fb_stat(xIN_Enable  := enIN_State = enState.StateAUTO,
        xIN_Waiting := fb_Pnp.xOUT_Wait,
        xIN_Running := (fb_Pnp.iOUT_Step >= ST180_Pnp_e.START) AND
                       (fb_Pnp.iOUT_Step <= ST180_Pnp_e.DONE),
        // Since we use a mover system, a cycle is done when we are waiting on a mover
        xIN_Done := fb_Pnp.iOUT_Step = ST180_Pnp_e.waitOnMover);

(*******************************************************************)
(* Mover reset flags *)
(*******************************************************************)

(*******************************************************************)
(* OUTPUT *)
(*******************************************************************)
xOUT_InitDone := fb_Pnp.xOUT_InitDone;
xOUT_Ready    := fb_Pnp.xOUT_Ready;
xOUT_Done     := fb_Pnp.xOUT_Done;
xOUT_ErrFlag  := fb_Pnp.xOUT_ErrFlag;
xOUT_Wait     := fb_Pnp.xOUT_Wait;
xOUT_AlarmST  := xOUT_ErrFlag;

(*******************************************************************)
(* Bausteinaufruf Error Station *)
(*******************************************************************)
// POU_ERR_VORLAGE(xIN_QUIT:=xIN_Quit , pstrArIN_ALARM:=ADR(HMI.strArALARM[1]));

(* % of completion of the process *)
PROPERTY iCompletionPC : INT
GET
iCompletionPC := THIS^.fb_Pnp.iOUT_ProcessCompletion;
END_GET
END_PROPERTY

PROPERTY ProcessExecution : ProcessExecution_e
GET
ProcessExecution := THIS^._ProcessExecution;
END_GET
SET
THIS^._ProcessExecution := ProcessExecution;
END_SET
END_PROPERTY

PROPERTY xBusy : BOOL
GET
xBusy := THIS^.fb_Pnp.xOUT_Busy;
END_GET
SET
END_SET
END_PROPERTY

PROPERTY xDone : BOOL
GET
xDone := THIS^.fb_Pnp.xOUT_Ready OR THIS^.fb_Pnp.xOUT_Done;
END_GET
END_PROPERTY

PROPERTY xMoverPathFree : BOOL
GET
xMoverPathFree := THIS^.fb_Pnp.xOUT_MoverFree OR THIS^.fb_Pnp.xOUT_Ready OR THIS^.fb_Pnp.xOUT_Done;
END_GET
END_PROPERTY

PROPERTY xMoverShouldLeave : BOOL
GET
xMoverShouldLeave := THIS^.fb_Pnp.iOUT_Step = ST180_Pnp_e.SYNC_MOVER_LEAVE;
END_GET
END_PROPERTY

END_FUNCTION_BLOCK

// ---- POUs/20_AUTO/ST180/FB_ABL_180_Pnp.TcPOU
FUNCTION_BLOCK FB_ABL_180_Pnp
(****************************************************************************************)
(*	TITEL				laden kristall- Modul	    										*)
(*	Status				ungetestet                         								*)
(*	Beschrieb:			Ablaufbeschreibung												*)
(*																						*)
(*	Steps:	self-explained using enum													*)
(***********************************Revisionen*******************************************)
(*	see github blames																	*)
(****************************************************************************************)

VAR_INPUT
    xIN_Reset       : BOOL;          // Schrittkette zurücksetzen 
    xIN_Init        : BOOL;          // Initialisieren
    xIN_Quit        : BOOL;          // Fehler quittieren 
    xIN_Start       : BOOL;          // Startbefehl
    xIN_Sperre      : BOOL;          // FB Sperren 
    xIN_NextStep    : BOOL;          // Nächsten Schritt ausführen 
    xIN_AlarmAktiv  : BOOL;          // Anlage hat Alarm
    xIN_DryCycle    : BOOL;          // Fahren ohne Teile
    xIN_RestartCYCL : BOOL;          // Zyklus erneut starten im STEP: END: LEERFAHREN
    enIN_State      : enState;       // Status Anlage
    tIN_Timeout     : TIME := T#10s; // Timout

    pxFG_Freigabe : POINTER TO BOOL; //Freigabe von Station

    // Application specific
    Mover              : REFERENCE TO FB_Mover;
    xIN_PceReadyToPick : BOOL; // the piece(s) is/are ready to picked
END_VAR
VAR_OUTPUT
    (* standart Ausgänge *)
    xOUT_ErrFlag  : BOOL;        // Error Flag 
    xOUT_Busy     : BOOL;        // Baustein befindet sich im Ablauf 
    xOUT_Done     : BOOL;        // Baustein hat den Ablauf beendet 		
    xOUT_Ready    : BOOL;        // Ready to begin: should be the same state as done	
    xOUT_Timeout  : BOOL;        // Timeout FB 
    xOUT_InitDone : BOOL;        // initialisierung fertig
    xOUT_Wait     : BOOL;        // Wartet auf Bedingung
    iOUT_Step     : ST180_Pnp_e; // Aktueller Schritt 
    sOUT_Step     : STRING;      // Aktueller Schritt but in string format
    bOUT_Error    : BYTE;        // Fehlernummer

    iOUT_ProcessCompletion : INT;  //process completion: express in % (0-100)
    xOUT_MoverFree         : BOOL; // The mover is free to move

END_VAR
VAR
    (* Standard *)
    (* Schritt *)
    iLastStep : ST180_Pnp_e; // Merker letzter Schritt 
    iPreStep  : ST180_Pnp_e; // Schritt zurück nach Alarm 
    iAktStep  : ST180_Pnp_e; // aktueller Schritt

    // Trigger Starten 
    rtSTART : R_TRIG;
    // Timer TimeOut 
    TON_Timeout : TON;

    (* Bausteine *)

    (* Spezial *)
    fb_axis180_01Y : FB_AxisLM_V1_1;
    fb_axis180_02Z : FB_AxisLM_V1_1;
    fb_axis180_10Z : FB_AxisLM_V1_1;

    fb_PnpHorAxis    : FB_LinearMotionMan;
    fb_PnpVerAxis_02 : FB_LinearMotionMan;
    fb_PnpVerAxis_10 : FB_LinearMotionMan;

    fb_simu_axis180_01Y : FB_Simu_AxisLM_V1_1;
    fb_simu_axis180_02Z : FB_Simu_AxisLM_V1_1;
    fb_simu_axis180_10Z : FB_Simu_AxisLM_V1_1;

    fb_griperLeft    : FB_ZylMo2El_V2_1;
    fb_griperRight   : FB_ZylMo2El_V2_1;
    simu_griperLeft  : FB_Simu_Zyl2Pos;
    simu_griperRight : FB_Simu_Zyl2Pos;
    fb_clampLeft     : FB_ZylMo2El_V2_1;
    fb_clampRight    : FB_ZylMo2El_V2_1;
    simu_clampLeft   : FB_Simu_Zyl2Pos;
    simu_clampRight  : FB_Simu_Zyl2Pos;

END_VAR
VAR CONSTANT
    PNP_SIMULATION : BOOL := FALSE; // Set to TRUE to simulate this part of the program
END_VAR

(*******************************************************************)
(* Trigger  *)
(*******************************************************************)
(* Zurücksetzen *)
IF xIN_RESET THEN
    iPreStep  := ST180_Pnp_e.RESET;
    iOUT_Step := ST180_Pnp_e.RESET;
END_IF;

(* Error Quittieren *)
IF (bOUT_Error <> 0) AND xIN_Quit THEN
    xOUT_ErrFlag := FALSE;
    bOUT_Error   := 0;
    iOUT_Step    := iPreStep;
END_IF;

(*******************************************************************)
(* Timer *)
(*******************************************************************)
TON_Timeout(IN := xIN_NextStep AND (iLastStep = iOUT_Step) (*todo FG *) ,
            PT := tIN_Timeout);

(*******************************************************************)
(* Bausteine *)
(*******************************************************************)
fb_PnpHorAxis(config          := _20_AUTO.recipe.linearAxis[LinearAxis_e.ST180_01Y],
              xIN_Init        := enIN_State = enState.StateINIT,
              xIN_Reset       := xIN_Reset,
              lrIN_CurrPos    := fb_axis180_01Y.rOUT_ActPos,
              lrIN_Delta_mm   := 1.0,
              iIN_CurrentStep := iOUT_Step,
              iIN_moveNumber  := ST180_PnpHorPos_e._max);

fb_simu_axis180_01Y(xIN_Enable          := PNP_SIMULATION AND CONST.USE_SIMULATION,
                    bIN_AxisCntr        := fb_axis180_01Y.bOUT_AxisCntr,
                    wIN_AxisState       := ST180_Axis.axis180_01Y.wState,
                    udiIN_HomingTime_ms := 2000,
                    pIN_axisSimu        := ADR(SIMU.axis_ref[Axis_e.ST180_01Y]),
                    pIN_axisHW          := ADR(ST180_Axis.axis180_01Y.axis),
                    rIN_PosActual       := ST180_Axis.axis180_01Y.rActPos,
                    rIN_PosMax          := ST180_Axis.const180_01Y.POS_MAX,
                    rIN_PosMin          := ST180_Axis.const180_01Y.POS_MIN,
                    rIN_PixMax          := 100,
                    rIN_PixMin          := 0);

fb_axis180_01Y(enIN_State       := enIN_State,
               parIN_Buttons    := ADR(AXIS.btTeachArAxis[Axis_e.ST180_01Y]),
               xIN_DisButtons   := FALSE,
               xIN_Quit         := xIN_Quit,
               xIN_PARAMok      := TRUE, (*TODO*)
               xIN_FREE         := TRUE,
               xIN_FREE_HOME    := TRUE,
               rIN_POSMIN       := ST180_Axis.const180_01Y.POS_MIN,
               rIN_POSMAX       := ST180_Axis.const180_01Y.POS_MAX,
               rIN_VELOMAX      := ST180_Axis.const180_01Y.VELO_MAX,
               rIN_VELOMANU     := ST180_Axis.const180_01Y.VELO_MANU,
               rIN_VELOOPEN     := ST180_Axis.const180_01Y.VELO_MANU / 4,
               rIN_JogInc       := AXIS.rTeachIncAxis,
               xIN_Execute      := fb_PnpHorAxis.xOUT_Execute,
               xIN_Relative     := FALSE,
               xIN_STOP         := FALSE,
               xIN_OFF          := FALSE,
               rIN_Position     := TO_REAL(fb_PnpHorAxis.OUT_MoveProfile.lrPosition),
               rIN_Velocity     := TO_REAL(fb_PnpHorAxis.OUT_MoveProfile.lrVelocity),
               rIN_Acceleration := TO_REAL(fb_PnpHorAxis.OUT_MoveProfile.lrAccel),
               rIN_Deceleration := TO_REAL(fb_PnpHorAxis.OUT_MoveProfile.lrDecel),
               rIN_Jerk         := TO_REAL(fb_PnpHorAxis.OUT_MoveProfile.lrJerk),
               rIN_PosManu      := TO_REAL(_20_AUTO.recipe.linearAxis[LinearAxis_e.ST180_01Y]
                                               .movesList[AXIS.bTeachPos[Axis_e.ST180_01Y]].lrPosition),
               rIN_VeloJogManu := TO_REAL(Axis.rJogVelo_pc),
               xIN_Home        := ST180_Pnp_e.Init_HomeHorizontal = iOUT_Step,
               xIN_Reset       := (ST180_Pnp_e.RESET = iOUT_Step) OR xIN_Reset,
               // The simu fb gives the hardware state when we are not in simu
               wAxisState    := fb_simu_axis180_01Y.wOUT_AxisState,
               bOUT_AxisCntr => st180_axis.axis180_01Y.bCtrlHi,
               rOUT_ActPos   => st180_axis.axis180_01Y.rActPos,
               axisIN_REF    := fb_simu_axis180_01Y.pOUT_axisRef^);

fb_PnpVerAxis_02(config          := _20_AUTO.recipe.linearAxis[LinearAxis_e.ST180_02Z],
                 xIN_Init        := enIN_State = enState.StateINIT,
                 xIN_Reset       := xIN_Reset,
                 lrIN_CurrPos    := fb_axis180_02Z.rOUT_ActPos,
                 lrIN_Delta_mm   := 2.50,
                 iIN_CurrentStep := iOUT_Step,
                 iIN_moveNumber  := ST180_PnpVerPos_e._max);

fb_simu_axis180_02Z(xIN_Enable          := PNP_SIMULATION AND CONST.USE_SIMULATION,
                    bIN_AxisCntr        := fb_axis180_02Z.bOUT_AxisCntr,
                    wIN_AxisState       := ST180_Axis.axis180_02Z.wState,
                    udiIN_HomingTime_ms := 2000,
                    pIN_axisSimu        := ADR(SIMU.axis_ref[Axis_e.ST180_02Z]),
                    pIN_axisHW          := ADR(ST180_Axis.axis180_02Z.axis),
                    rIN_PosActual       := ST180_Axis.axis180_02Z.rActPos,
                    rIN_PosMax          := ST180_Axis.const180_02Z.POS_MAX,
                    rIN_PosMin          := ST180_Axis.const180_02Z.POS_MIN,
                    rIN_PixMax          := 100,
                    rIN_PixMin          := 0);

fb_axis180_02Z(enIN_State       := enIN_State,
               parIN_Buttons    := ADR(AXIS.btTeachArAxis[Axis_e.ST180_02Z]),
               xIN_DisButtons   := FALSE,
               xIN_Quit         := xIN_Quit,
               xIN_PARAMok      := TRUE,
               xIN_FREE         := TRUE,
               xIN_FREE_HOME    := TRUE,
               rIN_POSMIN       := ST180_Axis.const180_02Z.POS_MIN,
               rIN_POSMAX       := ST180_Axis.const180_02Z.POS_MAX,
               rIN_VELOMAX      := ST180_Axis.const180_02Z.VELO_MAX,
               rIN_VELOMANU     := ST180_Axis.const180_02Z.VELO_MANU,
               rIN_VELOOPEN     := ST180_Axis.const180_02Z.POS_MAX / 4,
               rIN_JogInc       := AXIS.rTeachIncAxis,
               xIN_Execute      := fb_PnpVerAxis_02.xOUT_Execute,
               xIN_Relative     := FALSE,
               xIN_STOP         := FALSE,
               xIN_OFF          := FALSE,
               rIN_Position     := TO_REAL(fb_PnpVerAxis_02.OUT_MoveProfile.lrPosition),
               rIN_Velocity     := TO_REAL(fb_PnpVerAxis_02.OUT_MoveProfile.lrVelocity),
               rIN_Acceleration := TO_REAL(fb_PnpVerAxis_02.OUT_MoveProfile.lrAccel),
               rIN_Deceleration := TO_REAL(fb_PnpVerAxis_02.OUT_MoveProfile.lrDecel),
               rIN_Jerk         := TO_REAL(fb_PnpVerAxis_02.OUT_MoveProfile.lrJerk),
               rIN_PosManu      := TO_REAL(_20_AUTO.recipe.linearAxis[LinearAxis_e.ST180_02Z]
                                               .movesList[AXIS.bTeachPos[Axis_e.ST180_02Z]].lrPosition),
               rIN_VeloJogManu := TO_REAL(Axis.rJogVelo_pc),
               xIN_Home        := ST180_Pnp_e.Init_HomeVertical_02 = iOUT_Step,
               xIN_Reset       := (ST180_Pnp_e.RESET = iOUT_Step) OR xIN_Reset,
               wAxisState      := fb_simu_axis180_02Z.wOUT_AxisState,
               bOUT_AxisCntr   => ST180_Axis.axis180_02Z.bCtrlHi,
               rOUT_ActPos     => ST180_Axis.axis180_02Z.rActPos,
               axisIN_REF      := fb_simu_axis180_02Z.pOUT_axisRef^);

fb_PnpVerAxis_10(config          := _20_AUTO.recipe.linearAxis[LinearAxis_e.ST180_10Z],
                 xIN_Init        := enIN_State = enState.StateINIT,
                 xIN_Reset       := xIN_Reset,
                 lrIN_CurrPos    := fb_axis180_10Z.rOUT_ActPos,
                 lrIN_Delta_mm   := 1.0,
                 iIN_CurrentStep := iOUT_Step,
                 iIN_moveNumber  := ST180_PnpVerPos_e._max);

fb_simu_axis180_10Z(xIN_Enable          := PNP_SIMULATION AND CONST.USE_SIMULATION,
                    bIN_AxisCntr        := fb_axis180_10Z.bOUT_AxisCntr,
                    wIN_AxisState       := ST180_Axis.axis180_10Z.wState,
                    udiIN_HomingTime_ms := 2000,
                    pIN_axisSimu        := ADR(SIMU.axis_ref[Axis_e.ST180_10Z]),
                    pIN_axisHW          := ADR(ST180_Axis.axis180_10Z.axis),
                    rIN_PosActual       := ST180_Axis.axis180_10Z.rActPos,
                    rIN_PosMax          := ST180_Axis.const180_10Z.POS_MAX,
                    rIN_PosMin          := ST180_Axis.const180_10Z.POS_MIN,
                    rIN_PixMax          := 100,
                    rIN_PixMin          := 0);

fb_axis180_10Z(enIN_State       := enIN_State,
               parIN_Buttons    := ADR(AXIS.btTeachArAxis[Axis_e.ST180_10Z]),
               xIN_DisButtons   := FALSE,
               xIN_Quit         := xIN_Quit,
               xIN_PARAMok      := TRUE,
               xIN_FREE         := TRUE,
               xIN_FREE_HOME    := TRUE,
               rIN_POSMIN       := ST180_Axis.const180_10Z.POS_MIN,
               rIN_POSMAX       := ST180_Axis.const180_10Z.POS_MAX,
               rIN_VELOMAX      := ST180_Axis.const180_10Z.VELO_MAX,
               rIN_VELOMANU     := ST180_Axis.const180_10Z.VELO_MANU,
               rIN_VELOOPEN     := ST180_Axis.const180_10Z.POS_MAX / 4,
               rIN_JogInc       := AXIS.rTeachIncAxis,
               xIN_Execute      := fb_PnpVerAxis_10.xOUT_Execute,
               xIN_Relative     :=,
               xIN_STOP         :=,
               xIN_OFF          :=,
               rIN_Position     := TO_REAL(fb_PnpVerAxis_10.OUT_MoveProfile.lrPosition),
               rIN_Velocity     := TO_REAL(fb_PnpVerAxis_10.OUT_MoveProfile.lrVelocity),
               rIN_Acceleration := TO_REAL(fb_PnpVerAxis_10.OUT_MoveProfile.lrAccel),
               rIN_Deceleration := TO_REAL(fb_PnpVerAxis_10.OUT_MoveProfile.lrDecel),
               rIN_Jerk         := TO_REAL(fb_PnpVerAxis_10.OUT_MoveProfile.lrJerk),
               rIN_PosManu      := TO_REAL(_20_AUTO.recipe.linearAxis[LinearAxis_e.ST180_10Z]
                                               .movesList[AXIS.bTeachPos[Axis_e.ST180_10Z]].lrPosition),
               rIN_VeloJogManu := TO_REAL(Axis.rJogVelo_pc),
               xIN_Home        := ST180_Pnp_e.Init_HomeVertical_10 = iOUT_Step,
               xIN_Reset       := (ST180_Pnp_e.RESET = iOUT_Step) OR xIN_Reset,
               wAxisState      := fb_simu_axis180_10Z.wOUT_AxisState,
               bOUT_AxisCntr   => ST180_Axis.axis180_10Z.bCtrlHi,
               rOUT_ActPos     => ST180_Axis.axis180_10Z.rActPos,
               axisIN_REF      := fb_simu_axis180_10Z.pOUT_axisRef^);

//////////////////////////////////
fb_griperLeft(xIN_Reset    := xIN_Reset OR (ST180_Pnp_e.RESET = iOUT_Step),
              xIN_Quit     := xIN_Quit,
              xIN_Manu     := enState.StateMANU = enIN_State,
              pbtIN_Button := ADR(HMI.btManuCylinders[StationList_e.ST180][1]),
              xIN_GS       := simu_griperLeft.xOUT_inGS,
              xIN_AS       := simu_griperLeft.xOUT_inAS,
              xIN_FREE     := TRUE,
              xINtoGS      := _20_AUTO.recipe.st180.xUseVerLeft AND ST180_Pnp_e.close_griper_pick_piece = iOUT_Step,
              xINtoAS      := ST180_Pnp_e.open_griper_put_piece = iOUT_Step,
              tIN_ErrAS    := DINT_TO_TIME(_20_AUTO.recipe.cylinder2Pos[StationList_e.ST180]
                                               [ST180_Cylinders_e.Greifer_Patrone_Links].toAS_alarm_time),
              tIN_ErrGS := DINT_TO_TIME(_20_AUTO.recipe.cylinder2Pos[StationList_e.ST180]
                                            [ST180_Cylinders_e.Greifer_Patrone_Links].toGS_alarm_time),
              tIN_WaitAS := DINT_TO_TIME(_20_AUTO.recipe.cylinder2Pos[StationList_e.ST180]
                                             [ST180_Cylinders_e.Greifer_Patrone_Links].toAS_wait_time),
              tIN_WaitGS := DINT_TO_TIME(_20_AUTO.recipe.cylinder2Pos[StationList_e.ST180]
                                             [ST180_Cylinders_e.Greifer_Patrone_Links].toGS_wait_time));

simu_griperLeft(xIN_Enable := PNP_SIMULATION AND CONST.USE_SIMULATION,
                xIN_inGS   := IO_BOX.I9100_ST180_greifer_patrone_links_zu,
                xIN_inAS   := IO_BOX.I9101_ST180_greifer_patrone_links_offen,
                xIN_valve  := fb_griperLeft.xOUT_VALVE,
                tIN_GS_ms  := 200,  //ms
                tIN_AS_ms  := 200); //ms

fb_griperRight(xIN_Reset    := xIN_Reset OR (ST180_Pnp_e.RESET = iOUT_Step),
               xIN_Quit     := xIN_Quit,
               xIN_Manu     := enState.StateMANU = enIN_State,
               pbtIN_Button := ADR(HMI.btManuCylinders[StationList_e.ST180][2]),
               xIN_GS       := simu_griperRight.xOUT_inGS,
               xIN_AS       := simu_griperRight.xOUT_inAS,
               xIN_FREE     := TRUE,
               xINtoGS      := _20_AUTO.recipe.st180.xUseVerRight AND ST180_Pnp_e.close_griper_pick_piece = iOUT_Step,
               xINtoAS      := ST180_Pnp_e.open_griper_put_piece = iOUT_Step,
               tIN_ErrAS    := DINT_TO_TIME(_20_AUTO.recipe.cylinder2Pos[StationList_e.ST180]
                                                [ST180_Cylinders_e.Greifer_Patrone_Rechts].toAS_alarm_time),
               tIN_ErrGS := DINT_TO_TIME(_20_AUTO.recipe.cylinder2Pos[StationList_e.ST180]
                                             [ST180_Cylinders_e.Greifer_Patrone_Rechts].toGS_alarm_time),
               tIN_WaitAS := DINT_TO_TIME(_20_AUTO.recipe.cylinder2Pos[StationList_e.ST180]
                                              [ST180_Cylinders_e.Greifer_Patrone_Rechts].toAS_wait_time),
               tIN_WaitGS := DINT_TO_TIME(_20_AUTO.recipe.cylinder2Pos[StationList_e.ST180]
                                              [ST180_Cylinders_e.Greifer_Patrone_Rechts].toGS_wait_time));

simu_griperRight(xIN_Enable := PNP_SIMULATION AND CONST.USE_SIMULATION,
                 xIN_inGS   := IO_BOX.I9102_ST180_greifer_patrone_rechts_zu,
                 xIN_inAS   := IO_BOX.I9103_ST180_greifer_patrone_rechts_offen,
                 xIN_valve  := fb_griperRight.xOUT_VALVE,
                 tIN_GS_ms  := 200,  //ms
                 tIN_AS_ms  := 200); //ms

fb_clampLeft(xIN_Reset    := xIN_Reset OR (ST180_Pnp_e.RESET = iOUT_Step),
             xIN_Quit     := xIN_Quit,
             xIN_Manu     := enState.StateMANU = enIN_State,
             pbtIN_Button := ADR(HMI.btManuCylinders[StationList_e.ST180][3]),
             xIN_GS       := simu_clampLeft.xOUT_inGS,
             xIN_AS       := simu_clampLeft.xOUT_inAS,
             xIN_FREE     := TRUE,
             xINtoGS      := ST180_Pnp_e.clamp_up_to_rest_position = iOUT_Step,
             xINtoAS      := _20_AUTO.recipe.st180.xUseVerLeft AND
                             (ST180_Pnp_e.clamp_down_maintain_piece = iOUT_Step),
             tIN_ErrAS := DINT_TO_TIME(_20_AUTO.recipe.cylinder2Pos[StationList_e.ST180]
                                           [ST180_Cylinders_e.Niederhalter_Deckel_Links].toAS_alarm_time),
             tIN_ErrGS := DINT_TO_TIME(_20_AUTO.recipe.cylinder2Pos[StationList_e.ST180]
                                           [ST180_Cylinders_e.Niederhalter_Deckel_Links].toGS_alarm_time),
             tIN_WaitAS := DINT_TO_TIME(_20_AUTO.recipe.cylinder2Pos[StationList_e.ST180]
                                            [ST180_Cylinders_e.Niederhalter_Deckel_Links].toAS_wait_time),
             tIN_WaitGS := DINT_TO_TIME(_20_AUTO.recipe.cylinder2Pos[StationList_e.ST180]
                                            [ST180_Cylinders_e.Niederhalter_Deckel_Links].toGS_wait_time));

simu_clampLeft(xIN_Enable := PNP_SIMULATION AND CONST.USE_SIMULATION,
               xIN_inGS   := IO_BOX.I9104_ST180_niederhalter_deckel_links_oben,
               xIN_inAS   := NOT IO_BOX.I9104_ST180_niederhalter_deckel_links_oben,
               xIN_valve  := fb_clampLeft.xOUT_VALVE,
               tIN_GS_ms  := 200,  //ms
               tIN_AS_ms  := 200); //ms

fb_clampRight(xIN_Reset    := xIN_Reset OR (ST180_Pnp_e.RESET = iOUT_Step),
              xIN_Quit     := xIN_Quit,
              xIN_Manu     := enState.StateMANU = enIN_State,
              pbtIN_Button := ADR(HMI.btManuCylinders[StationList_e.ST180][4]),
              xIN_GS       := simu_clampRight.xOUT_inGS,
              xIN_AS       := simu_clampRight.xOUT_inAS,
              xIN_FREE     := TRUE,
              xINtoGS      := ST180_Pnp_e.clamp_up_to_rest_position = iOUT_Step,
              xINtoAS      := _20_AUTO.recipe.st180.xUseVerRight AND
                              (ST180_Pnp_e.clamp_down_maintain_piece = iOUT_Step),
              tIN_ErrAS := DINT_TO_TIME(_20_AUTO.recipe.cylinder2Pos[StationList_e.ST180]
                                            [ST180_Cylinders_e.Niederhalter_Deckel_Rechts].toAS_alarm_time),
              tIN_ErrGS := DINT_TO_TIME(_20_AUTO.recipe.cylinder2Pos[StationList_e.ST180]
                                            [ST180_Cylinders_e.Niederhalter_Deckel_Rechts].toGS_alarm_time),
              tIN_WaitAS := DINT_TO_TIME(_20_AUTO.recipe.cylinder2Pos[StationList_e.ST180]
                                             [ST180_Cylinders_e.Niederhalter_Deckel_Rechts].toAS_wait_time),
              tIN_WaitGS := DINT_TO_TIME(_20_AUTO.recipe.cylinder2Pos[StationList_e.ST180]
                                             [ST180_Cylinders_e.Niederhalter_Deckel_Rechts].toGS_wait_time));

simu_clampRight(xIN_Enable := PNP_SIMULATION AND CONST.USE_SIMULATION,
                xIN_inGS   := IO_BOX.I9106_ST180_niederhalter_deckel_rechts_oben,
                xIN_inAS   := NOT IO_BOX.I9106_ST180_niederhalter_deckel_rechts_oben,
                xIN_valve  := fb_clampRight.xOUT_VALVE,
                tIN_GS_ms  := 200,  // ms
                tIN_AS_ms  := 200); // ms

(*******************************************************************)
(* OUTPUTS *)
(*******************************************************************)
// Error Flag 
xOUT_ErrFlag := (bOUT_Error <> 0) OR (ST180_Pnp_e.ERROR = iOUT_Step);
// Baustein befindet sich im Ablauf 
xOUT_Busy := (iOUT_Step > ST180_Pnp_e.READY) AND (iOUT_Step < ST180_Pnp_e.DONE);
// Baustein hat den Ablauf beendet
xOUT_Done := (iOUT_Step = ST180_Pnp_e.DONE);
// Process ready
xOUT_Ready := (iOUT_Step = ST180_Pnp_e.READY) OR (iOUT_Step = ST180_Pnp_e.hor_move_to_extraction_pipe);
// Timeout FB 				 		
xOUT_Timeout := TON_Timeout.Q;
// Itialisierung fertig			
xOUT_InitDone := (iOUT_Step = ST180_Pnp_e.READY) OR
                 (iOUT_Step = ST180_Pnp_e.hor_move_to_extraction_pipe) OR
                 (iOUT_Step = ST180_Pnp_e.DONE);

// Aktueller Schritt			
iOUT_Step := iOUT_Step; //Im Ablauf gesetzt		
sOUT_Step := TO_STRING(iOUT_Step);
//Fehlernummer	 
bOUT_Error := bOUT_Error; //Im Ablauf/FB gesetzt	
(* Warte (alle Schritte wo auf FG oder Teile gewartet wird) *)
xOUT_Wait := (iOUT_Step = ST180_Pnp_e.DONE) OR
             (iOUT_Step = ST180_Pnp_e.READY) OR
             (iOUT_Step = ST180_Pnp_e.START) OR
             (iOUT_Step = ST180_Pnp_e.waitOnMover) OR
             (iOUT_Step = ST180_Pnp_e.SYNC_MOVER_LEAVE);

xOUT_MoverFree := NOT (iOUT_Step >= ST180_Pnp_e.MOVER_NEEDED_OP AND iOUT_Step < ST180_Pnp_e.MOVER_FREE_OP) AND
                  (iOUT_Step >= ST180_Pnp_e.READY) AND
                  (iOUT_Step < ST180_Pnp_e.ERROR);

iOUT_ProcessCompletion := F_GetPercent_2(iOUT_Step,
                                         ST180_Pnp_e.lift_piece_and_down_to_pick,
                                         ST180_Pnp_e.take_out_piece_and_put_down_lifter,
                                         ST180_Pnp_e.hor_move_to_extraction_pipe,
                                         ST180_Pnp_e.hor_to_track_pos);

// TODO Valve should not be set when we are in simulation !
IO_BOX.Q5400_14_ST180_greifer_patrone_links :=
    fb_griperLeft.xOUT_VALVE AND NOT (PNP_SIMULATION AND CONST.USE_SIMULATION);

IO_BOX.Q5401_14_ST180_greifer_patrone_rechts :=
    fb_griperRight.xOUT_VALVE AND NOT (PNP_SIMULATION AND CONST.USE_SIMULATION);

IO_BOX.Q5402_14_ST180_niederhalter_deckel_links :=
    fb_clampLeft.xOUT_VALVE AND NOT (PNP_SIMULATION AND CONST.USE_SIMULATION);

IO_BOX.Q5403_14_ST180_Niederhalter_deckel_rechts :=
    fb_clampRight.xOUT_VALVE AND NOT (PNP_SIMULATION AND CONST.USE_SIMULATION);

// safety pneumatics
IO_BOX.Q5408_14_ST180_Break_axis_02Z := NOT fb_simu_axis180_02Z.pIN_axisHW^.Status.Error AND
                                        _02_SAFETY.xOUT_ESout AND
                                        _02_SAFETY.xOUT_MonOut AND
                                        NOT (PNP_SIMULATION AND CONST.USE_SIMULATION);

(*******************************************************************)
(* Ablauf *)
(*******************************************************************)

(* Sperren *)
IF xIN_Sperre THEN
    iPreStep  := ST180_Pnp_e.RESET;
    iOUT_Step := ST180_Pnp_e.RESET;
    RETURN;
END_IF;

(* Schritt Merker *)
IF iAktStep <> iOUT_Step THEN
    iLastStep := iAktStep;
    iAktStep  := iOUT_Step;
END_IF

(* START *)
rtSTART(CLK := xIN_Start);

IF 0 = bOUT_Error THEN
    IF fb_axis180_01Y.xOUT_ErrFlag THEN
        bOUT_Error := 11;
    ELSIF fb_axis180_02Z.xOUT_ErrFlag THEN
        bOUT_Error := 12;
    ELSIF fb_axis180_10Z.xOUT_ErrFlag THEN
        bOUT_Error := 13;
    ELSIF fb_griperLeft.xOUT_ErrFlag THEN
        bOUT_Error := 14;
    ELSIF fb_griperRight.xOUT_ErrFlag THEN
        bOUT_Error := 15;
    ELSIF fb_clampLeft.xOUT_ErrFlag THEN
        bOUT_Error := 16;
    ELSIF fb_clampRight.xOUT_ErrFlag THEN
        bOUT_Error := 17;
    END_IF
ELSIF iOUT_Step < ST180_Pnp_e.ERROR THEN
    iOUT_Step := ST180_Pnp_e.ERROR;
END_IF

(*******************************************************************)
(* Schrittkette  *)
(*******************************************************************)
CASE iOUT_Step OF

(***** RESET *****)
ST180_Pnp_e.RESET: (* Schritt 0-99 *)
    //Initialisierungen
    //Start Init Ablauf
    IF xIN_Init THEN
        iOUT_Step := ST180_Pnp_e.INIT;
        //Start Manu Ablauf
    ELSIF enIN_State = StateMANU AND xIN_NextStep THEN
        iOUT_Step := ST180_Pnp_e.INIT;
    END_IF;

(***** INIT *****)
ST180_Pnp_e.INIT: (* Grundstellung ? *)
    IF fb_axis180_10Z.xOUT_HOMED THEN
        iOUT_Step := ST180_Pnp_e.Init_Vertical_10_Down;
    ELSE
        iOUT_Step := ST180_Pnp_e.Init_HomeVertical_10;
    END_IF

ST180_Pnp_e.Init_HomeVertical_10:
    IF fb_axis180_10Z.xOUT_HOMED THEN
        iOUT_Step := ST180_Pnp_e.Init_Vertical_10_Down;
    END_IF

ST180_Pnp_e.Init_Vertical_10_Down:
    IF fb_PnpVerAxis_10.MoveTo(ST180_PnpHorPos_e.GS).xOUT_InPos THEN
        IF fb_axis180_02Z.xOUT_HOMED THEN
            iOUT_Step := ST180_Pnp_e.Init_Vertical_02_up;
        ELSE
            iOUT_Step := ST180_Pnp_e.Init_HomeVertical_02;
        END_IF
    END_IF

ST180_Pnp_e.Init_HomeVertical_02:
    IF fb_axis180_02Z.xOUT_HOMED THEN
        iOUT_Step := ST180_Pnp_e.Init_Vertical_02_up;
    END_IF

ST180_Pnp_e.Init_Vertical_02_up:
    IF fb_griperLeft.xIN_GS OR fb_griperRight.xIN_GS THEN
        IF fb_PnpVerAxis_02.MoveTo(ST180_PnpVerPos_e.up_after_unload).xOUT_InPos THEN
            IF fb_axis180_01Y.xOUT_HOMED THEN
                iOUT_Step := ST180_Pnp_e.Init_HorizontalToTrack;
            ELSE
                iOUT_Step := ST180_Pnp_e.Init_HomeHorizontal;
            END_IF
        END_IF
    ELSE
        IF fb_PnpVerAxis_02.MoveTo(ST180_PnpVerPos_e.up_waiting_mover).xOUT_InPos THEN
            IF fb_axis180_01Y.xOUT_HOMED THEN
                iOUT_Step := ST180_Pnp_e.Init_HorizontalToTrack;
            ELSE
                iOUT_Step := ST180_Pnp_e.Init_HomeHorizontal;
            END_IF
        END_IF
    END_IF

ST180_Pnp_e.Init_HomeHorizontal:
    IF fb_axis180_01Y.xOUT_HOMED THEN
        iOUT_Step := ST180_Pnp_e.Init_HorizontalToTrack;
    END_IF

ST180_Pnp_e.Init_HorizontalToTrack:
    IF fb_PnpHorAxis.MoveTo(ST180_PnpHorPos_e.GS).xOUT_InPos THEN
        iOUT_Step := ST180_Pnp_e.Init_check_if_pces_handled;
    END_IF

ST180_Pnp_e.Init_check_if_pces_handled:
    IF (NOT _20_AUTO.recipe.st180.xUseVerLeft AND fb_griperLeft.xOUT_inGS) OR
       (NOT _20_AUTO.recipe.st180.xUseVerRight AND fb_griperRight.xOUT_inGS) THEN
        // ERROR: a piece is present in an unused gripper
        bOUT_Error := 1;
        iOUT_Step  := ST180_Pnp_e.ERROR;

    ELSIF _20_AUTO.recipe.st180.xUseVerLeft AND
          NOT fb_griperLeft.xOUT_inGS AND
          _20_AUTO.recipe.st180.xUseVerRight AND
          fb_griperRight.xOUT_inGS THEN
        // ERROR:  Initialisation failed. A piece is missing in the left griper.
        bOUT_Error := 2;
        iOUT_Step  := ST180_Pnp_e.ERROR;

    ELSIF _20_AUTO.recipe.st180.xUseVerLeft AND
          fb_griperLeft.xOUT_inGS AND
          _20_AUTO.recipe.st180.xUseVerRight AND
          NOT fb_griperRight.xOUT_inGS THEN
        // ERROR:  Initialisation failed. A piece is missing in the right griper.
        bOUT_Error := 3;
        iOUT_Step  := ST180_Pnp_e.ERROR;

    ELSIF NOT fb_griperLeft.xOUT_inGS AND NOT fb_griperRight.xOUT_inGS THEN
        iOUT_Step := ST180_Pnp_e.READY;

    ELSE
        iOUT_Step := ST180_Pnp_e.hor_move_to_extraction_pipe;
    END_IF

(***** READY / INIT DONE *****)
ST180_Pnp_e.READY:    (* Start AUTO:END:LEER:STEP *)
    IF xIN_Start THEN //IF rtSTART.Q THEN
        iOUT_Step := ST180_Pnp_e.START;
    END_IF

(***** START  ZYKLISCH *****)
ST180_Pnp_e.START: (*  *)
    IF xIN_NextStep AND pxFG_Freigabe^ THEN
        iOUT_Step := ST180_Pnp_e.waitOnMover;
    END_IF;

ST180_Pnp_e.waitOnMover:
    IF xIN_NextStep AND __ISVALIDREF(Mover) OR HMI.bArForceCyclusState[StationList_e.ST180] THEN
        IF Mover.IsPieceBad() THEN
            iOUT_Step := ST180_Pnp_e.lift_piece_and_down_to_pick;
        ELSE
            iOUT_Step := ST180_Pnp_e.SYNC_MOVER_LEAVE;
        END_IF
    END_IF

ST180_Pnp_e.lift_piece_and_down_to_pick:
    IF xIN_NextStep AND
       fb_PnpVerAxis_02.MoveTo(ST180_PnpVerPos_e.down_empty).xOUT_InPos AND
       fb_PnpVerAxis_10.MoveTo(ST180_PnpHorPos_e.AS).xOUT_InPos THEN
        iOUT_Step := ST180_Pnp_e.close_griper_pick_piece;
    END_IF

ST180_Pnp_e.close_griper_pick_piece:
    IF xIN_NextStep AND
       (NOT _20_AUTO.recipe.st180.xUseVerLeft OR fb_griperLeft.xOUT_inGS) AND
       (NOT _20_AUTO.recipe.st180.xUseVerRight OR fb_griperRight.xOUT_inGS) THEN
        iOUT_Step := ST180_Pnp_e.clamp_down_maintain_piece;
    END_IF

ST180_Pnp_e.clamp_down_maintain_piece:
    IF xIN_NextStep AND
       (NOT _20_AUTO.recipe.st180.xUseVerLeft OR fb_clampLeft.xOUT_inAS) AND
       (NOT _20_AUTO.recipe.st180.xUseVerRight OR fb_clampRight.xOUT_inAS) THEN
        iOUT_Step := ST180_Pnp_e.take_out_piece_and_put_down_lifter;
    END_IF

ST180_Pnp_e.take_out_piece_and_put_down_lifter:
    IF xIN_NextStep AND
       fb_PnpVerAxis_02.MoveTo(ST180_PnpVerPos_e.up_full).xOUT_InPos AND
       fb_PnpVerAxis_10.MoveTo(ST180_PnpHorPos_e.GS).xOUT_InPos THEN
        iOUT_Step := ST180_Pnp_e.SYNC_MOVER_LEAVE;

        IF __ISVALIDREF(Mover) THEN
            Mover.UnloadPieces();
        END_IF
    END_IF

ST180_Pnp_e.SYNC_MOVER_LEAVE:
    // The mover needs to be taken by MoverMan
    IF NOT __ISVALIDREF(Mover) THEN
        IF (NOT _20_AUTO.recipe.st180.xUseVerLeft OR fb_griperLeft.xIN_GS) AND
           (NOT _20_AUTO.recipe.st180.xUseVerRight OR fb_griperRight.xIN_GS) THEN
            iOUT_Step := ST180_Pnp_e.hor_move_to_extraction_pipe;
        ELSE
            iOUT_Step := ST180_Pnp_e.DONE;
        END_IF
    END_IF

ST180_Pnp_e.hor_move_to_extraction_pipe:
    IF xIN_NextStep AND fb_PnpHorAxis.MoveTo(ST180_PnpHorPos_e.AS).xOUT_InPos THEN
        iOUT_Step := ST180_Pnp_e.ver_down_in_pipe;
    END_IF

ST180_Pnp_e.ver_down_in_pipe:
    IF xIN_NextStep AND fb_PnpVerAxis_02.MoveTo(ST180_PnpVerPos_e.down_full).xOUT_InPos THEN
        iOUT_Step := ST180_Pnp_e.clamp_up_to_rest_position;
    END_IF

ST180_Pnp_e.clamp_up_to_rest_position:
    IF xIN_NextStep AND
       (NOT _20_AUTO.recipe.st180.xUseVerLeft OR fb_clampLeft.xOUT_inGS) AND
       (NOT _20_AUTO.recipe.st180.xUseVerRight OR fb_clampRight.xOUT_inGS) THEN
        iOUT_Step := ST180_Pnp_e.open_griper_put_piece;
    END_IF

ST180_Pnp_e.open_griper_put_piece:
    IF xIN_NextStep AND
       (NOT _20_AUTO.recipe.st180.xUseVerLeft OR fb_griperLeft.xOUT_inAS) AND
       (NOT _20_AUTO.recipe.st180.xUseVerRight OR fb_griperRight.xOUT_inAS) THEN
        // We check if we need to move up or not, this is to avoid colision with 
        iOUT_Step := ST180_Pnp_e.ver_up_empty;
    END_IF

ST180_Pnp_e.ver_up_empty:
    IF xIN_NextStep AND fb_PnpVerAxis_02.MoveTo(ST180_PnpVerPos_e.up_after_unload).xOUT_InPos THEN
        iOUT_Step := ST180_Pnp_e.hor_to_track_pos;
    END_IF

ST180_Pnp_e.hor_to_track_pos:
    IF xIN_NextStep AND fb_PnpHorAxis.MoveTo(ST180_PnpHorPos_e.GS).xOUT_InPos THEN
        iOUT_Step := ST180_Pnp_e.ver_down_waiting_for_mover;
    END_IF

ST180_Pnp_e.ver_down_waiting_for_mover:
    IF xIN_NextStep AND fb_PnpVerAxis_02.MoveTo(ST180_PnpVerPos_e.up_waiting_mover).xOUT_InPos THEN
        iOUT_Step := ST180_Pnp_e.DONE;
    END_IF

(***** DONE *****)
ST180_Pnp_e.DONE: (* Letzter Schritt  *)
    IF NOT xIN_AlarmAktiv THEN
        //AUTO
        IF (enIN_State = StateAUTO) AND xIN_RestartCYCL THEN
            iOUT_Step := ST180_Pnp_e.START;
            //STEP / END / LEERFAHREN restart
        ELSIF (enIN_State < StateAUTO) AND (enIN_State >= enState.StateSTEP) AND xIN_RestartCYCL THEN
            iOUT_Step := ST180_Pnp_e.START;
            //STEP / END / LEERFAHREN fertig
        ELSIF (enIN_State = StateREADY) THEN
            iOUT_Step := ST180_Pnp_e.READY;
        END_IF;
    END_IF;

(************ ERROR *************)
ST180_Pnp_e.ERROR: (* ERROR *) ;

END_CASE;

END_FUNCTION_BLOCK

// ---- POUs/20_AUTO/ST185/FB_AUT_185.TcPOU
FUNCTION_BLOCK FB_AUT_185 EXTENDS FB_AUT_ABSTRACT
(****************************************************************************)
(*	POU_AUT_zxx			Bausteinaufrufe Station	zxx							*)
(*	Status				ungetestet											*)
(*  Version:			1.0													*)
(*	Beschrieb:																*)
(*																			*)
(*	Abläufe:			FB_ABLzxxA		Hauptablauf							*)
(*																			*)
(*																			*)
(* 	25.09.2019/Dj															*)
(****************************************************************************)
(*	dd.mm.yyyy   KZ    x.y			Beschrieb								*)
(****************************************************************************)
VAR_INPUT
    (* spezifische Eingänge *)

END_VAR
VAR_OUTPUT
    (* spezifische Ausgänge *)

END_VAR
VAR
    (* Bausteine *)
    fb_Pnp    : FB_ABL_185_Pnp;

    fb_stat : FB_AUT_Statistics;

END_VAR

(*******************************************************************)
(* Timer *)
(*******************************************************************)

(*******************************************************************)
(* Flanken / Merker *)
(*******************************************************************)
//MANU CYCLE
IF (enIN_State = StateMANU) AND xIN_ManuCycle THEN
    xManuCycle := TRUE;
END_IF;

IF (enIN_State <> StateMANU) OR xOUT_Done THEN
    xManuCycle := FALSE;
END_IF

//NEXT STEP
xNextStep := (enIN_State > StateSTEP) OR
             ((enIN_State = StateSTEP) AND xIN_Step) OR
             ((enIN_State = StateMANU) AND xManuCycle);

//RESET
xReset := (enIN_State < StateREADY) AND (enIN_State <> StateINIT) AND NOT xManuCycle;

(*******************************************************************)
(* Bausteinaufrufe Abläufe *)
(*******************************************************************)

xRelease := MAIN.MoverMan.IsProcessUsed(THIS^);

fb_Pnp(xIN_Reset          := xReset,
       xIN_Init           := xIN_Init,
       xIN_Quit           := xIN_Quit,
       xIN_Start          := enIN_State >= enState.StateLEER AND xRelease,
       xIN_Sperre         := NOT xIN_On,
       xIN_NextStep       := xNextStep,
       xIN_AlarmAktiv     := xIN_AlarmAktiv,
       xIN_DryCycle       := xIN_DryCycle,
       xIN_RestartCYCL    := enIN_State >= enState.StateLEER,
       enIN_State         := enIN_State,
       tIN_Timeout        := tIN_Timeout,
       pxFG_Freigabe      := ADR(xRelease),
       Mover              := THIS^.Mover,
       xIN_PceReadyToPick := TRUE);

fb_stat(xIN_Enable  := enIN_State = enState.StateAUTO,
        xIN_Waiting := fb_Pnp.xOUT_Wait,
        xIN_Running := (fb_Pnp.iOUT_Step >= ST185_Pnp_e.START) AND
                       (fb_Pnp.iOUT_Step <= ST185_Pnp_e.DONE),
        // Since we use a mover system, a cycle is done when we are waiting on a mover
        xIN_Done := fb_Pnp.iOUT_Step = ST185_Pnp_e.waitOnMover);

(*******************************************************************)
(* Mover reset flags *)
(*******************************************************************)

(*******************************************************************)
(* OUTPUT *)
(*******************************************************************)
xOUT_InitDone := fb_Pnp.xOUT_InitDone;
xOUT_Ready    := fb_Pnp.xOUT_Ready;
xOUT_Done     := fb_Pnp.xOUT_Done;
xOUT_ErrFlag  := fb_Pnp.xOUT_ErrFlag;
xOUT_Wait     := fb_Pnp.xOUT_Wait;
xOUT_AlarmST  := xOUT_ErrFlag;

(*******************************************************************)
(* Bausteinaufruf Error Station *)
(*******************************************************************)
// POU_ERR_VORLAGE(xIN_QUIT:=xIN_Quit , pstrArIN_ALARM:=ADR(HMI.strArALARM[1]));

(* % of completion of the process *)
PROPERTY iCompletionPC : INT
GET
iCompletionPC := THIS^.fb_Pnp.iOUT_ProcessCompletion;
END_GET
END_PROPERTY

PROPERTY ProcessExecution : ProcessExecution_e
GET
ProcessExecution := THIS^._ProcessExecution;
END_GET
SET
THIS^._ProcessExecution := ProcessExecution;
END_SET
END_PROPERTY

PROPERTY xBusy : BOOL
GET
xBusy := THIS^.fb_Pnp.xOUT_Busy;
END_GET
SET
END_SET
END_PROPERTY

PROPERTY xDone : BOOL
GET
xDone := THIS^.fb_Pnp.xOUT_Ready OR THIS^.fb_Pnp.xOUT_Done;
END_GET
END_PROPERTY

PROPERTY xMoverPathFree : BOOL
GET
xMoverPathFree := THIS^.fb_Pnp.xOUT_MoverFree OR THIS^.fb_Pnp.xOUT_Ready OR THIS^.fb_Pnp.xOUT_Done;
END_GET
END_PROPERTY

PROPERTY xMoverShouldLeave : BOOL
GET
xMoverShouldLeave := THIS^.fb_Pnp.iOUT_Step = ST185_Pnp_e.SYNC_MOVER_LEAVE;
END_GET
END_PROPERTY

END_FUNCTION_BLOCK

// ---- POUs/20_AUTO/ST185/FB_ABL_185_Pnp.TcPOU
FUNCTION_BLOCK FB_ABL_185_Pnp
(****************************************************************************************)
(*	TITEL				laden kristall- Modul	    										*)
(*	Status				ungetestet                         								*)
(*	Beschrieb:			Ablaufbeschreibung												*)
(*																						*)
(*	Steps:	self-explained using enum													*)
(***********************************Revisionen*******************************************)
(*	see github blames																	*)
(****************************************************************************************)

VAR_INPUT
    xIN_Reset       : BOOL;          // Schrittkette zurücksetzen 
    xIN_Init        : BOOL;          // Initialisieren
    xIN_Quit        : BOOL;          // Fehler quittieren 
    xIN_Start       : BOOL;          // Startbefehl
    xIN_Sperre      : BOOL;          // FB Sperren 
    xIN_NextStep    : BOOL;          // Nächsten Schritt ausführen 
    xIN_AlarmAktiv  : BOOL;          // Anlage hat Alarm
    xIN_DryCycle    : BOOL;          // Fahren ohne Teile
    xIN_RestartCYCL : BOOL;          // Zyklus erneut starten im STEP: END: LEERFAHREN
    enIN_State      : enState;       // Status Anlage
    tIN_Timeout     : TIME := T#10s; // Timout

    pxFG_Freigabe : POINTER TO BOOL; //Freigabe von Station

    // Application specific
    Mover              : REFERENCE TO FB_Mover;
    xIN_PceReadyToPick : BOOL; // the piece(s) is/are ready to picked
END_VAR
VAR_OUTPUT
    (* standart Ausgänge *)
    xOUT_ErrFlag  : BOOL;        // Error Flag 
    xOUT_Busy     : BOOL;        // Baustein befindet sich im Ablauf 
    xOUT_Done     : BOOL;        // Baustein hat den Ablauf beendet 		
    xOUT_Ready    : BOOL;        // Ready to begin: should be the same state as done	
    xOUT_Timeout  : BOOL;        // Timeout FB 
    xOUT_InitDone : BOOL;        // initialisierung fertig
    xOUT_Wait     : BOOL;        // Wartet auf Bedingung
    iOUT_Step     : ST185_Pnp_e; // Aktueller Schritt 
    sOUT_Step     : STRING;      // Aktueller Schritt but in string format
    bOUT_Error    : BYTE;        // Fehlernummer

    iOUT_ProcessCompletion : INT;  //process completion: express in % (0-100)
    xOUT_MoverFree         : BOOL; // The mover is free to move

END_VAR
VAR
    (* Standard *)
    (* Schritt *)
    iLastStep : ST185_Pnp_e; // Merker letzter Schritt 
    iPreStep  : ST185_Pnp_e; // Schritt zurück nach Alarm 
    iAktStep  : ST185_Pnp_e; // aktueller Schritt

    // Trigger Starten 
    rtSTART : R_TRIG;
    // Timer TimeOut 
    TON_Timeout : TON;

    (* Bausteine *)

    (* Spezial *)
    fb_axis185_01Y : FB_AxisLM_V1_1;
    fb_axis185_02Z : FB_AxisLM_V1_1;
    fb_axis185_10Z : FB_AxisLM_V1_1;

    fb_PnpHorAxis    : FB_LinearMotionMan;
    fb_PnpVerAxis_02 : FB_LinearMotionMan;
    fb_PnpVerAxis_10 : FB_LinearMotionMan;

    fb_simu_axis185_01Y : FB_Simu_AxisLM_V1_1;
    fb_simu_axis185_02Z : FB_Simu_AxisLM_V1_1;
    fb_simu_axis185_10Z : FB_Simu_AxisLM_V1_1;

    fb_griperLeft    : FB_ZylMo2El_V2_1;
    fb_griperRight   : FB_ZylMo2El_V2_1;
    simu_griperLeft  : FB_Simu_Zyl2Pos;
    simu_griperRight : FB_Simu_Zyl2Pos;
    fb_clampLeft     : FB_ZylMo2El_V2_1;
    fb_clampRight    : FB_ZylMo2El_V2_1;
    simu_clampLeft   : FB_Simu_Zyl2Pos;
    simu_clampRight  : FB_Simu_Zyl2Pos;

    arrLrAvgCycleTime : ARRAY[0..AVERAGE_ARRAY_SIZE - 1] OF LREAL;
    lrStartCycleTime  : UDINT;
    indexAvgArray     : INT := 0;
    sumAvgArray       : LREAL;
    i                 : INT;

END_VAR
VAR CONSTANT
    PNP_SIMULATION : BOOL := FALSE; // Set to TRUE to simulate this part of the program

    AVERAGE_ARRAY_SIZE : INT := 16;
END_VAR

(*******************************************************************)
(* Trigger  *)
(*******************************************************************)
(* Zurücksetzen *)
IF xIN_RESET THEN
    iPreStep  := ST185_Pnp_e.RESET;
    iOUT_Step := ST185_Pnp_e.RESET;
END_IF;

(* Error Quittieren *)
IF (bOUT_Error <> 0) AND xIN_Quit THEN
    xOUT_ErrFlag := FALSE;
    bOUT_Error   := 0;
    iOUT_Step    := iPreStep;
END_IF;

(*******************************************************************)
(* Timer *)
(*******************************************************************)
TON_Timeout(IN := xIN_NextStep AND (iLastStep = iOUT_Step) (*todo FG *) ,
            PT := tIN_Timeout);

(*******************************************************************)
(* Bausteine *)
(*******************************************************************)
fb_PnpHorAxis(config          := _20_AUTO.recipe.linearAxis[LinearAxis_e.ST185_01Y],
              xIN_Init        := enIN_State = enState.StateINIT,
              xIN_Reset       := xIN_Reset,
              lrIN_CurrPos    := fb_axis185_01Y.rOUT_ActPos,
              lrIN_Delta_mm   := 0.5,
              iIN_CurrentStep := iOUT_Step,
              iIN_moveNumber  := ST185_PnpHorPos_e._max);

fb_simu_axis185_01Y(xIN_Enable          := PNP_SIMULATION AND CONST.USE_SIMULATION,
                    bIN_AxisCntr        := fb_axis185_01Y.bOUT_AxisCntr,
                    wIN_AxisState       := ST185_Axis.axis185_01Y.wState,
                    udiIN_HomingTime_ms := 2000,
                    pIN_axisSimu        := ADR(SIMU.axis_ref[Axis_e.ST185_01Y]),
                    pIN_axisHW          := ADR(ST185_Axis.axis185_01Y.axis),
                    rIN_PosActual       := ST185_Axis.axis185_01Y.rActPos,
                    rIN_PosMax          := ST185_Axis.const185_01Y.POS_MAX,
                    rIN_PosMin          := ST185_Axis.const185_01Y.POS_MIN,
                    rIN_PixMax          := 100,
                    rIN_PixMin          := 0);

fb_axis185_01Y(enIN_State       := enIN_State,
               parIN_Buttons    := ADR(AXIS.btTeachArAxis[Axis_e.ST185_01Y]),
               xIN_DisButtons   := FALSE,
               xIN_Quit         := xIN_Quit,
               xIN_PARAMok      := TRUE, (*TODO*)
               xIN_FREE         := TRUE,
               xIN_FREE_HOME    := TRUE,
               rIN_POSMIN       := ST185_Axis.const185_01Y.POS_MIN,
               rIN_POSMAX       := ST185_Axis.const185_01Y.POS_MAX,
               rIN_VELOMAX      := ST185_Axis.const185_01Y.VELO_MAX,
               rIN_VELOMANU     := ST185_Axis.const185_01Y.VELO_MANU,
               rIN_VELOOPEN     := ST185_Axis.const185_01Y.VELO_MANU / 4,
               rIN_JogInc       := AXIS.rTeachIncAxis,
               xIN_Execute      := fb_PnpHorAxis.xOUT_Execute,
               xIN_Relative     := FALSE,
               xIN_STOP         := FALSE,
               xIN_OFF          := FALSE,
               rIN_Position     := TO_REAL(fb_PnpHorAxis.OUT_MoveProfile.lrPosition),
               rIN_Velocity     := TO_REAL(fb_PnpHorAxis.OUT_MoveProfile.lrVelocity),
               rIN_Acceleration := TO_REAL(fb_PnpHorAxis.OUT_MoveProfile.lrAccel),
               rIN_Deceleration := TO_REAL(fb_PnpHorAxis.OUT_MoveProfile.lrDecel),
               rIN_Jerk         := TO_REAL(fb_PnpHorAxis.OUT_MoveProfile.lrJerk),
               rIN_PosManu      := TO_REAL(_20_AUTO.recipe.linearAxis[LinearAxis_e.ST185_01Y]
                                               .movesList[AXIS.bTeachPos[Axis_e.ST185_01Y]].lrPosition),
               rIN_VeloJogManu := TO_REAL(Axis.rJogVelo_pc),
               xIN_Home        := ST185_Pnp_e.Init_HomeHorizontal = iOUT_Step,
               xIN_Reset       := (ST185_Pnp_e.RESET = iOUT_Step) OR xIN_Reset,
               // The simu fb gives the hardware state when we are not in simu
               wAxisState    := fb_simu_axis185_01Y.wOUT_AxisState,
               bOUT_AxisCntr => st185_axis.axis185_01Y.bCtrlHi,
               rOUT_ActPos   => st185_axis.axis185_01Y.rActPos,
               axisIN_REF    := fb_simu_axis185_01Y.pOUT_axisRef^);

fb_PnpVerAxis_02(config          := _20_AUTO.recipe.linearAxis[LinearAxis_e.ST185_02Z],
                 xIN_Init        := enIN_State = enState.StateINIT,
                 xIN_Reset       := xIN_Reset,
                 lrIN_CurrPos    := fb_axis185_02Z.rOUT_ActPos,
                 lrIN_Delta_mm   := 2.50,
                 iIN_CurrentStep := iOUT_Step,
                 iIN_moveNumber  := ST185_PnpVerPos_e._max);

fb_simu_axis185_02Z(xIN_Enable          := PNP_SIMULATION AND CONST.USE_SIMULATION,
                    bIN_AxisCntr        := fb_axis185_02Z.bOUT_AxisCntr,
                    wIN_AxisState       := ST185_Axis.axis185_02Z.wState,
                    udiIN_HomingTime_ms := 2000,
                    pIN_axisSimu        := ADR(SIMU.axis_ref[Axis_e.ST185_02Z]),
                    pIN_axisHW          := ADR(ST185_Axis.axis185_02Z.axis),
                    rIN_PosActual       := ST185_Axis.axis185_02Z.rActPos,
                    rIN_PosMax          := ST185_Axis.const185_02Z.POS_MAX,
                    rIN_PosMin          := ST185_Axis.const185_02Z.POS_MIN,
                    rIN_PixMax          := 100,
                    rIN_PixMin          := 0);

fb_axis185_02Z(enIN_State       := enIN_State,
               parIN_Buttons    := ADR(AXIS.btTeachArAxis[Axis_e.ST185_02Z]),
               xIN_DisButtons   := FALSE,
               xIN_Quit         := xIN_Quit,
               xIN_PARAMok      := TRUE,
               xIN_FREE         := TRUE,
               xIN_FREE_HOME    := TRUE,
               rIN_POSMIN       := ST185_Axis.const185_02Z.POS_MIN,
               rIN_POSMAX       := ST185_Axis.const185_02Z.POS_MAX,
               rIN_VELOMAX      := ST185_Axis.const185_02Z.VELO_MAX,
               rIN_VELOMANU     := ST185_Axis.const185_02Z.VELO_MANU,
               rIN_VELOOPEN     := ST185_Axis.const185_02Z.POS_MAX / 4,
               rIN_JogInc       := AXIS.rTeachIncAxis,
               xIN_Execute      := fb_PnpVerAxis_02.xOUT_Execute,
               xIN_Relative     := FALSE,
               xIN_STOP         := FALSE,
               xIN_OFF          := FALSE,
               rIN_Position     := TO_REAL(fb_PnpVerAxis_02.OUT_MoveProfile.lrPosition),
               rIN_Velocity     := TO_REAL(fb_PnpVerAxis_02.OUT_MoveProfile.lrVelocity),
               rIN_Acceleration := TO_REAL(fb_PnpVerAxis_02.OUT_MoveProfile.lrAccel),
               rIN_Deceleration := TO_REAL(fb_PnpVerAxis_02.OUT_MoveProfile.lrDecel),
               rIN_Jerk         := TO_REAL(fb_PnpVerAxis_02.OUT_MoveProfile.lrJerk),
               rIN_PosManu      := TO_REAL(_20_AUTO.recipe.linearAxis[LinearAxis_e.ST185_02Z]
                                               .movesList[AXIS.bTeachPos[Axis_e.ST185_02Z]].lrPosition),
               rIN_VeloJogManu := TO_REAL(Axis.rJogVelo_pc),
               xIN_Home        := ST185_Pnp_e.Init_HomeVertical_02 = iOUT_Step,
               xIN_Reset       := (ST185_Pnp_e.RESET = iOUT_Step) OR xIN_Reset,
               wAxisState      := fb_simu_axis185_02Z.wOUT_AxisState,
               bOUT_AxisCntr   => ST185_Axis.axis185_02Z.bCtrlHi,
               rOUT_ActPos     => ST185_Axis.axis185_02Z.rActPos,
               axisIN_REF      := fb_simu_axis185_02Z.pOUT_axisRef^);

fb_PnpVerAxis_10(config          := _20_AUTO.recipe.linearAxis[LinearAxis_e.ST185_10Z],
                 xIN_Init        := enIN_State = enState.StateINIT,
                 xIN_Reset       := xIN_Reset,
                 lrIN_CurrPos    := fb_axis185_10Z.rOUT_ActPos,
                 lrIN_Delta_mm   := 1.0,
                 iIN_CurrentStep := iOUT_Step,
                 iIN_moveNumber  := ST185_PnpVerPos_e._max);

fb_simu_axis185_10Z(xIN_Enable          := PNP_SIMULATION AND CONST.USE_SIMULATION,
                    bIN_AxisCntr        := fb_axis185_10Z.bOUT_AxisCntr,
                    wIN_AxisState       := ST185_Axis.axis185_10Z.wState,
                    udiIN_HomingTime_ms := 2000,
                    pIN_axisSimu        := ADR(SIMU.axis_ref[Axis_e.ST185_10Z]),
                    pIN_axisHW          := ADR(ST185_Axis.axis185_10Z.axis),
                    rIN_PosActual       := ST185_Axis.axis185_10Z.rActPos,
                    rIN_PosMax          := ST185_Axis.const185_10Z.POS_MAX,
                    rIN_PosMin          := ST185_Axis.const185_10Z.POS_MIN,
                    rIN_PixMax          := 100,
                    rIN_PixMin          := 0);

fb_axis185_10Z(enIN_State       := enIN_State,
               parIN_Buttons    := ADR(AXIS.btTeachArAxis[Axis_e.ST185_10Z]),
               xIN_DisButtons   := FALSE,
               xIN_Quit         := xIN_Quit,
               xIN_PARAMok      := TRUE,
               xIN_FREE         := TRUE,
               xIN_FREE_HOME    := TRUE,
               rIN_POSMIN       := ST185_Axis.const185_10Z.POS_MIN,
               rIN_POSMAX       := ST185_Axis.const185_10Z.POS_MAX,
               rIN_VELOMAX      := ST185_Axis.const185_10Z.VELO_MAX,
               rIN_VELOMANU     := ST185_Axis.const185_10Z.VELO_MANU,
               rIN_VELOOPEN     := ST185_Axis.const185_10Z.POS_MAX / 4,
               rIN_JogInc       := AXIS.rTeachIncAxis,
               xIN_Execute      := fb_PnpVerAxis_10.xOUT_Execute,
               xIN_Relative     :=,
               xIN_STOP         :=,
               xIN_OFF          :=,
               rIN_Position     := TO_REAL(fb_PnpVerAxis_10.OUT_MoveProfile.lrPosition),
               rIN_Velocity     := TO_REAL(fb_PnpVerAxis_10.OUT_MoveProfile.lrVelocity),
               rIN_Acceleration := TO_REAL(fb_PnpVerAxis_10.OUT_MoveProfile.lrAccel),
               rIN_Deceleration := TO_REAL(fb_PnpVerAxis_10.OUT_MoveProfile.lrDecel),
               rIN_Jerk         := TO_REAL(fb_PnpVerAxis_10.OUT_MoveProfile.lrJerk),
               rIN_PosManu      := TO_REAL(_20_AUTO.recipe.linearAxis[LinearAxis_e.ST185_10Z]
                                               .movesList[AXIS.bTeachPos[Axis_e.ST185_10Z]].lrPosition),
               rIN_VeloJogManu := TO_REAL(Axis.rJogVelo_pc),
               xIN_Home        := ST185_Pnp_e.Init_HomeVertical_10 = iOUT_Step,
               xIN_Reset       := (ST185_Pnp_e.RESET = iOUT_Step) OR xIN_Reset,
               wAxisState      := fb_simu_axis185_10Z.wOUT_AxisState,
               bOUT_AxisCntr   => ST185_Axis.axis185_10Z.bCtrlHi,
               rOUT_ActPos     => ST185_Axis.axis185_10Z.rActPos,
               axisIN_REF      := fb_simu_axis185_10Z.pOUT_axisRef^);

//////////////////////////////////
fb_griperLeft(xIN_Reset    := xIN_Reset OR (ST185_Pnp_e.RESET = iOUT_Step),
              xIN_Quit     := xIN_Quit,
              xIN_Manu     := enState.StateMANU = enIN_State,
              pbtIN_Button := ADR(HMI.btManuCylinders[StationList_e.ST185][1]),
              xIN_GS       := simu_griperLeft.xOUT_inGS,
              xIN_AS       := simu_griperLeft.xOUT_inAS,
              xIN_FREE     := TRUE,
              xINtoGS      := _20_AUTO.recipe.st185.xUseVerLeft AND ST185_Pnp_e.close_griper_pick_piece = iOUT_Step,
              xINtoAS      := ST185_Pnp_e.open_griper_put_piece = iOUT_Step,
              tIN_ErrAS    := DINT_TO_TIME(_20_AUTO.recipe.cylinder2Pos[StationList_e.ST185]
                                               [ST185_Cylinders_e.Greifer_Patrone_Links].toAS_alarm_time),
              tIN_ErrGS := DINT_TO_TIME(_20_AUTO.recipe.cylinder2Pos[StationList_e.ST185]
                                            [ST185_Cylinders_e.Greifer_Patrone_Links].toGS_alarm_time),
              tIN_WaitAS := DINT_TO_TIME(_20_AUTO.recipe.cylinder2Pos[StationList_e.ST185]
                                             [ST185_Cylinders_e.Greifer_Patrone_Links].toAS_wait_time),
              tIN_WaitGS := DINT_TO_TIME(_20_AUTO.recipe.cylinder2Pos[StationList_e.ST185]
                                             [ST185_Cylinders_e.Greifer_Patrone_Links].toGS_wait_time));

simu_griperLeft(xIN_Enable := PNP_SIMULATION AND CONST.USE_SIMULATION,
                xIN_inGS   := IO_BOX.I9200_ST185_greifer_patrone_links_zu,
                xIN_inAS   := IO_BOX.I9201_ST185_greifer_patrone_links_offen,
                xIN_valve  := fb_griperLeft.xOUT_VALVE,
                tIN_GS_ms  := 200,  //ms
                tIN_AS_ms  := 200); //ms

fb_griperRight(xIN_Reset    := xIN_Reset OR (ST185_Pnp_e.RESET = iOUT_Step),
               xIN_Quit     := xIN_Quit,
               xIN_Manu     := enState.StateMANU = enIN_State,
               pbtIN_Button := ADR(HMI.btManuCylinders[StationList_e.ST185][2]),
               xIN_GS       := simu_griperRight.xOUT_inGS,
               xIN_AS       := simu_griperRight.xOUT_inAS,
               xIN_FREE     := TRUE,
               xINtoGS      := _20_AUTO.recipe.st185.xUseVerRight AND ST185_Pnp_e.close_griper_pick_piece = iOUT_Step,
               xINtoAS      := ST185_Pnp_e.open_griper_put_piece = iOUT_Step,
               tIN_ErrAS    := DINT_TO_TIME(_20_AUTO.recipe.cylinder2Pos[StationList_e.ST185]
                                                [ST185_Cylinders_e.Greifer_Patrone_Rechts].toAS_alarm_time),
               tIN_ErrGS := DINT_TO_TIME(_20_AUTO.recipe.cylinder2Pos[StationList_e.ST185]
                                             [ST185_Cylinders_e.Greifer_Patrone_Rechts].toGS_alarm_time),
               tIN_WaitAS := DINT_TO_TIME(_20_AUTO.recipe.cylinder2Pos[StationList_e.ST185]
                                              [ST185_Cylinders_e.Greifer_Patrone_Rechts].toAS_wait_time),
               tIN_WaitGS := DINT_TO_TIME(_20_AUTO.recipe.cylinder2Pos[StationList_e.ST185]
                                              [ST185_Cylinders_e.Greifer_Patrone_Rechts].toGS_wait_time));

simu_griperRight(xIN_Enable := PNP_SIMULATION AND CONST.USE_SIMULATION,
                 xIN_inGS   := IO_BOX.I9202_ST185_greifer_patrone_rechts_zu,
                 xIN_inAS   := IO_BOX.I9203_ST185_greifer_patrone_rechts_offen,
                 xIN_valve  := fb_griperRight.xOUT_VALVE,
                 tIN_GS_ms  := 200,  //ms
                 tIN_AS_ms  := 200); //ms

fb_clampLeft(xIN_Reset    := xIN_Reset OR (ST185_Pnp_e.RESET = iOUT_Step),
             xIN_Quit     := xIN_Quit,
             xIN_Manu     := enState.StateMANU = enIN_State,
             pbtIN_Button := ADR(HMI.btManuCylinders[StationList_e.ST185][3]),
             xIN_GS       := simu_clampLeft.xOUT_inGS,
             xIN_AS       := simu_clampLeft.xOUT_inAS,
             xIN_FREE     := TRUE,
             xINtoGS      := ST185_Pnp_e.clamp_up_to_rest_position = iOUT_Step,
             xINtoAS      := _20_AUTO.recipe.st185.xUseVerLeft AND
                             (ST185_Pnp_e.clamp_down_maintain_piece = iOUT_Step),
             tIN_ErrAS := DINT_TO_TIME(_20_AUTO.recipe.cylinder2Pos[StationList_e.ST185]
                                           [ST185_Cylinders_e.Niederhalter_Deckel_Links].toAS_alarm_time),
             tIN_ErrGS := DINT_TO_TIME(_20_AUTO.recipe.cylinder2Pos[StationList_e.ST185]
                                           [ST185_Cylinders_e.Niederhalter_Deckel_Links].toGS_alarm_time),
             tIN_WaitAS := DINT_TO_TIME(_20_AUTO.recipe.cylinder2Pos[StationList_e.ST185]
                                            [ST185_Cylinders_e.Niederhalter_Deckel_Links].toAS_wait_time),
             tIN_WaitGS := DINT_TO_TIME(_20_AUTO.recipe.cylinder2Pos[StationList_e.ST185]
                                            [ST185_Cylinders_e.Niederhalter_Deckel_Links].toGS_wait_time));

simu_clampLeft(xIN_Enable := PNP_SIMULATION AND CONST.USE_SIMULATION,
               xIN_inGS   := IO_BOX.I9204_ST185_niederhalter_deckel_links_oben,
               xIN_inAS   := NOT IO_BOX.I9204_ST185_niederhalter_deckel_links_oben,
               xIN_valve  := fb_clampLeft.xOUT_VALVE,
               tIN_GS_ms  := 200,  //ms
               tIN_AS_ms  := 200); //ms

fb_clampRight(xIN_Reset    := xIN_Reset OR (ST185_Pnp_e.RESET = iOUT_Step),
              xIN_Quit     := xIN_Quit,
              xIN_Manu     := enState.StateMANU = enIN_State,
              pbtIN_Button := ADR(HMI.btManuCylinders[StationList_e.ST185][4]),
              xIN_GS       := simu_clampRight.xOUT_inGS,
              xIN_AS       := simu_clampRight.xOUT_inAS,
              xIN_FREE     := TRUE,
              xINtoGS      := ST185_Pnp_e.clamp_up_to_rest_position = iOUT_Step,
              xINtoAS      := _20_AUTO.recipe.st185.xUseVerRight AND
                              (ST185_Pnp_e.clamp_down_maintain_piece = iOUT_Step),
              tIN_ErrAS := DINT_TO_TIME(_20_AUTO.recipe.cylinder2Pos[StationList_e.ST185]
                                            [ST185_Cylinders_e.Niederhalter_Deckel_Rechts].toAS_alarm_time),
              tIN_ErrGS := DINT_TO_TIME(_20_AUTO.recipe.cylinder2Pos[StationList_e.ST185]
                                            [ST185_Cylinders_e.Niederhalter_Deckel_Rechts].toGS_alarm_time),
              tIN_WaitAS := DINT_TO_TIME(_20_AUTO.recipe.cylinder2Pos[StationList_e.ST185]
                                             [ST185_Cylinders_e.Niederhalter_Deckel_Rechts].toAS_wait_time),
              tIN_WaitGS := DINT_TO_TIME(_20_AUTO.recipe.cylinder2Pos[StationList_e.ST185]
                                             [ST185_Cylinders_e.Niederhalter_Deckel_Rechts].toGS_wait_time));

simu_clampRight(xIN_Enable := PNP_SIMULATION AND CONST.USE_SIMULATION,
                xIN_inGS   := IO_BOX.I9206_ST185_niederhalter_deckel_rechts_oben,
                xIN_inAS   := NOT IO_BOX.I9206_ST185_niederhalter_deckel_rechts_oben,
                xIN_valve  := fb_clampRight.xOUT_VALVE,
                tIN_GS_ms  := 200,  // ms
                tIN_AS_ms  := 200); // ms

(*******************************************************************)
(* OUTPUTS *)
(*******************************************************************)
// Error Flag 
xOUT_ErrFlag := (bOUT_Error <> 0) OR (ST185_Pnp_e.ERROR = iOUT_Step);
// Baustein befindet sich im Ablauf 
xOUT_Busy := (iOUT_Step > ST185_Pnp_e.READY) AND (iOUT_Step < ST185_Pnp_e.DONE);
// Baustein hat den Ablauf beendet
xOUT_Done := (iOUT_Step = ST185_Pnp_e.DONE);
// Process ready
xOUT_Ready := (iOUT_Step = ST185_Pnp_e.READY) OR (iOUT_Step = ST185_Pnp_e.hor_move_to_extraction_pipe);
// Timeout FB 				 		
xOUT_Timeout := TON_Timeout.Q;
// Itialisierung fertig			
xOUT_InitDone := (iOUT_Step = ST185_Pnp_e.READY) OR
                 (iOUT_Step = ST185_Pnp_e.hor_move_to_extraction_pipe) OR
                 (iOUT_Step = ST185_Pnp_e.DONE);

// Aktueller Schritt			
iOUT_Step := iOUT_Step; //Im Ablauf gesetzt		
sOUT_Step := TO_STRING(iOUT_Step);
//Fehlernummer	 
bOUT_Error := bOUT_Error; //Im Ablauf/FB gesetzt	
(* Warte (alle Schritte wo auf FG oder Teile gewartet wird) *)
xOUT_Wait := (iOUT_Step = ST185_Pnp_e.DONE) OR
             (iOUT_Step = ST185_Pnp_e.READY) OR
             (iOUT_Step = ST185_Pnp_e.START) OR
             (iOUT_Step = ST185_Pnp_e.waitOnMover) OR
             (iOUT_Step = ST185_Pnp_e.SYNC_MOVER_LEAVE);

xOUT_MoverFree := NOT (iOUT_Step >= ST185_Pnp_e.MOVER_NEEDED_OP AND iOUT_Step < ST185_Pnp_e.MOVER_FREE_OP) AND
                  (iOUT_Step >= ST185_Pnp_e.READY) AND
                  (iOUT_Step < ST185_Pnp_e.ERROR);

iOUT_ProcessCompletion := F_GetPercent_2(iOUT_Step,
                                         ST185_Pnp_e.lift_piece_and_down_to_pick,
                                         ST185_Pnp_e.take_out_piece_and_put_down_lifter,
                                         ST185_Pnp_e.hor_move_to_extraction_pipe,
                                         ST185_Pnp_e.hor_to_track_pos);

// TODO Valve should not be set when we are in simulation !
IO_BOX.Q5404_14_ST185_greifer_patrone_links :=
    fb_griperLeft.xOUT_VALVE AND NOT (PNP_SIMULATION AND CONST.USE_SIMULATION);

IO_BOX.Q5405_14_ST185_greifer_patrone_rechts :=
    fb_griperRight.xOUT_VALVE AND NOT (PNP_SIMULATION AND CONST.USE_SIMULATION);

IO_BOX.Q5406_14_ST185_niederhalter_deckel_links :=
    fb_clampLeft.xOUT_VALVE AND NOT (PNP_SIMULATION AND CONST.USE_SIMULATION);

IO_BOX.Q5407_14_ST185_Niederhalter_deckel_rechts :=
    fb_clampRight.xOUT_VALVE AND NOT (PNP_SIMULATION AND CONST.USE_SIMULATION);

// safety pneumatics
IO_BOX.Q5409_14_ST185_Break_axis_02Z := NOT fb_simu_axis185_02Z.pIN_axisHW^.Status.Error AND
                                        _02_SAFETY.xOUT_ESout AND
                                        _02_SAFETY.xOUT_MonOut AND
                                        NOT (PNP_SIMULATION AND CONST.USE_SIMULATION);

OUT.Q102_ST185_entladen_ein :=
    (enIN_State >= enState.StateEND) AND
    ((iOUT_Step < ST185_Pnp_e.open_griper_put_piece) OR (iOUT_Step > ST185_Pnp_e.hor_to_track_pos)) AND
    NOT (PNP_SIMULATION AND CONST.USE_SIMULATION);

(*******************************************************************)
(* Ablauf *)
(*******************************************************************)

(* Sperren *)
IF xIN_Sperre THEN
    iPreStep  := ST185_Pnp_e.RESET;
    iOUT_Step := ST185_Pnp_e.RESET;
    RETURN;
END_IF;

(* Schritt Merker *)
IF iAktStep <> iOUT_Step THEN
    iLastStep := iAktStep;
    iAktStep  := iOUT_Step;
END_IF

(* START *)
rtSTART(CLK := xIN_Start);

IF 0 = bOUT_Error THEN
    IF fb_axis185_01Y.xOUT_ErrFlag THEN
        bOUT_Error := 11;
    ELSIF fb_axis185_02Z.xOUT_ErrFlag THEN
        bOUT_Error := 12;
    ELSIF fb_axis185_10Z.xOUT_ErrFlag THEN
        bOUT_Error := 13;
    ELSIF fb_griperLeft.xOUT_ErrFlag THEN
        bOUT_Error := 14;
    ELSIF fb_griperRight.xOUT_ErrFlag THEN
        bOUT_Error := 15;
    ELSIF fb_clampLeft.xOUT_ErrFlag THEN
        bOUT_Error := 16;
    ELSIF fb_clampRight.xOUT_ErrFlag THEN
        bOUT_Error := 17;
    END_IF
ELSIF iOUT_Step < ST185_Pnp_e.ERROR THEN
    iOUT_Step := ST185_Pnp_e.ERROR;
END_IF

(*******************************************************************)
(* Schrittkette  *)
(*******************************************************************)
CASE iOUT_Step OF

(***** RESET *****)
ST185_Pnp_e.RESET: (* Schritt 0-99 *)
    //Initialisierungen
    //Start Init Ablauf
    IF xIN_Init THEN
        iOUT_Step := ST185_Pnp_e.INIT;
        //Start Manu Ablauf
    ELSIF enIN_State = StateMANU AND xIN_NextStep THEN
        iOUT_Step := ST185_Pnp_e.INIT;
    END_IF;

(***** INIT *****)
ST185_Pnp_e.INIT: (* Grundstellung ? *)
    IF fb_axis185_10Z.xOUT_HOMED THEN
        iOUT_Step := ST185_Pnp_e.Init_Vertical_10_Down;
    ELSE
        iOUT_Step := ST185_Pnp_e.Init_HomeVertical_10;
    END_IF

ST185_Pnp_e.Init_HomeVertical_10:
    IF fb_axis185_10Z.xOUT_HOMED THEN
        iOUT_Step := ST185_Pnp_e.Init_Vertical_10_Down;
    END_IF

ST185_Pnp_e.Init_Vertical_10_Down:
    IF fb_PnpVerAxis_10.MoveTo(ST185_PnpHorPos_e.GS).xOUT_InPos THEN
        IF fb_axis185_02Z.xOUT_HOMED THEN
            iOUT_Step := ST185_Pnp_e.Init_Vertical_02_up;
        ELSE
            iOUT_Step := ST185_Pnp_e.Init_HomeVertical_02;
        END_IF
    END_IF

ST185_Pnp_e.Init_HomeVertical_02:
    IF fb_axis185_02Z.xOUT_HOMED THEN
        iOUT_Step := ST185_Pnp_e.Init_Vertical_02_up;
    END_IF

ST185_Pnp_e.Init_Vertical_02_up:
    IF fb_griperLeft.xIN_GS OR fb_griperRight.xIN_GS THEN
        IF fb_PnpVerAxis_02.MoveTo(ST185_PnpVerPos_e.up_after_unload).xOUT_InPos THEN
            IF fb_axis185_01Y.xOUT_HOMED THEN
                iOUT_Step := ST185_Pnp_e.Init_HorizontalToTrack;
            ELSE
                iOUT_Step := ST185_Pnp_e.Init_HomeHorizontal;
            END_IF
        END_IF
    ELSE
        IF fb_PnpVerAxis_02.MoveTo(ST185_PnpVerPos_e.up_waiting_mover).xOUT_InPos THEN
            IF fb_axis185_01Y.xOUT_HOMED THEN
                iOUT_Step := ST185_Pnp_e.Init_HorizontalToTrack;
            ELSE
                iOUT_Step := ST185_Pnp_e.Init_HomeHorizontal;
            END_IF
        END_IF
    END_IF

ST185_Pnp_e.Init_HomeHorizontal:
    IF fb_axis185_01Y.xOUT_HOMED THEN
        iOUT_Step := ST185_Pnp_e.Init_HorizontalToTrack;
    END_IF

ST185_Pnp_e.Init_HorizontalToTrack:
    IF fb_PnpHorAxis.MoveTo(ST185_PnpHorPos_e.GS).xOUT_InPos THEN
        iOUT_Step := ST185_Pnp_e.Init_check_if_pces_handled;
    END_IF

ST185_Pnp_e.Init_check_if_pces_handled:
    IF (NOT _20_AUTO.recipe.st185.xUseVerLeft AND fb_griperLeft.xOUT_inGS) OR
       (NOT _20_AUTO.recipe.st185.xUseVerRight AND fb_griperRight.xOUT_inGS) THEN
        // ERROR: a piece is present in an unused gripper
        bOUT_Error := 1;
        iOUT_Step  := ST185_Pnp_e.ERROR;

    ELSIF _20_AUTO.recipe.st185.xUseVerLeft AND
          NOT fb_griperLeft.xOUT_inGS AND
          _20_AUTO.recipe.st185.xUseVerRight AND
          fb_griperRight.xOUT_inGS THEN
        // ERROR:  Initialisation failed. A piece is missing in the left griper.
        bOUT_Error := 2;
        iOUT_Step  := ST185_Pnp_e.ERROR;

    ELSIF _20_AUTO.recipe.st185.xUseVerLeft AND
          fb_griperLeft.xOUT_inGS AND
          _20_AUTO.recipe.st185.xUseVerRight AND
          NOT fb_griperRight.xOUT_inGS THEN
        // ERROR:  Initialisation failed. A piece is missing in the right griper.
        bOUT_Error := 3;
        iOUT_Step  := ST185_Pnp_e.ERROR;

    ELSIF NOT fb_griperLeft.xOUT_inGS AND NOT fb_griperRight.xOUT_inGS THEN
        iOUT_Step := ST185_Pnp_e.READY;

    ELSE
        iOUT_Step := ST185_Pnp_e.hor_move_to_extraction_pipe;
    END_IF

(***** READY / INIT DONE *****)
ST185_Pnp_e.READY:    (* Start AUTO:END:LEER:STEP *)
    IF xIN_Start THEN //IF rtSTART.Q THEN
        iOUT_Step := ST185_Pnp_e.START;
    END_IF

(***** START  ZYKLISCH *****)
ST185_Pnp_e.START: (*  *)
    IF xIN_NextStep AND pxFG_Freigabe^ THEN
        lrStartCycleTime := GetTick();
        iOUT_Step        := ST185_Pnp_e.waitOnMover;
    END_IF;

ST185_Pnp_e.waitOnMover:
    IF xIN_NextStep AND __ISVALIDREF(Mover) OR HMI.bArForceCyclusState[StationList_e.ST185] THEN
        iOUT_Step := ST185_Pnp_e.lift_piece_and_down_to_pick;
    END_IF

ST185_Pnp_e.lift_piece_and_down_to_pick:
    IF xIN_NextStep AND
       fb_PnpVerAxis_02.MoveTo(ST185_PnpVerPos_e.down_empty).xOUT_InPos AND
       fb_PnpVerAxis_10.MoveTo(ST185_PnpHorPos_e.AS).xOUT_InPos THEN
        iOUT_Step := ST185_Pnp_e.close_griper_pick_piece;
    END_IF

ST185_Pnp_e.close_griper_pick_piece:
    IF xIN_NextStep AND
       (NOT _20_AUTO.recipe.st185.xUseVerLeft OR fb_griperLeft.xOUT_inGS) AND
       (NOT _20_AUTO.recipe.st185.xUseVerRight OR fb_griperRight.xOUT_inGS) THEN
        iOUT_Step := ST185_Pnp_e.clamp_down_maintain_piece;
    END_IF

ST185_Pnp_e.clamp_down_maintain_piece:
    IF xIN_NextStep AND
       (NOT _20_AUTO.recipe.st185.xUseVerLeft OR fb_clampLeft.xOUT_inAS) AND
       (NOT _20_AUTO.recipe.st185.xUseVerRight OR fb_clampRight.xOUT_inAS) THEN
        iOUT_Step := ST185_Pnp_e.take_out_piece_and_put_down_lifter;
    END_IF

ST185_Pnp_e.take_out_piece_and_put_down_lifter:
    IF xIN_NextStep AND
       fb_PnpVerAxis_02.MoveTo(ST185_PnpVerPos_e.up_full).xOUT_InPos AND
       fb_PnpVerAxis_10.MoveTo(ST185_PnpHorPos_e.GS).xOUT_InPos THEN
        iOUT_Step := ST185_Pnp_e.SYNC_MOVER_LEAVE;

        IF __ISVALIDREF(Mover) THEN
            Mover.UnloadPieces();
        END_IF
    END_IF

ST185_Pnp_e.SYNC_MOVER_LEAVE:
    // The mover needs to be taken by MoverMan
    IF NOT __ISVALIDREF(Mover) THEN
        iOUT_Step := ST185_Pnp_e.hor_move_to_extraction_pipe;
    END_IF

ST185_Pnp_e.hor_move_to_extraction_pipe:
    IF xIN_NextStep AND fb_PnpHorAxis.MoveTo(ST185_PnpHorPos_e.AS).xOUT_InPos THEN
        iOUT_Step := ST185_Pnp_e.ver_down_in_pipe;
    END_IF

ST185_Pnp_e.ver_down_in_pipe:
    IF xIN_NextStep AND fb_PnpVerAxis_02.MoveTo(ST185_PnpVerPos_e.down_full).xOUT_InPos THEN
        iOUT_Step := ST185_Pnp_e.clamp_up_to_rest_position;
    END_IF

ST185_Pnp_e.clamp_up_to_rest_position:
    IF xIN_NextStep AND
       (NOT _20_AUTO.recipe.st185.xUseVerLeft OR fb_clampLeft.xOUT_inGS) AND
       (NOT _20_AUTO.recipe.st185.xUseVerRight OR fb_clampRight.xOUT_inGS) THEN
        iOUT_Step := ST185_Pnp_e.open_griper_put_piece;
    END_IF

ST185_Pnp_e.open_griper_put_piece:
    IF xIN_NextStep AND
       (NOT _20_AUTO.recipe.st185.xUseVerLeft OR fb_griperLeft.xOUT_inAS) AND
       (NOT _20_AUTO.recipe.st185.xUseVerRight OR fb_griperRight.xOUT_inAS) THEN
        // We check if we need to move up or not, this is to avoid colision with 
        iOUT_Step := ST185_Pnp_e.ver_up_empty;
    END_IF

ST185_Pnp_e.ver_up_empty:
    IF xIN_NextStep AND fb_PnpVerAxis_02.MoveTo(ST185_PnpVerPos_e.up_after_unload).xOUT_InPos THEN
        iOUT_Step := ST185_Pnp_e.hor_to_track_pos;
    END_IF

ST185_Pnp_e.hor_to_track_pos:
    IF xIN_NextStep AND fb_PnpHorAxis.MoveTo(ST185_PnpHorPos_e.GS).xOUT_InPos THEN
        iOUT_Step := ST185_Pnp_e.ver_down_waiting_for_mover;
    END_IF

ST185_Pnp_e.ver_down_waiting_for_mover:
    IF xIN_NextStep AND fb_PnpVerAxis_02.MoveTo(ST185_PnpVerPos_e.up_waiting_mover).xOUT_InPos THEN

        arrLrAvgCycleTime[indexAvgArray] := GetTick() - lrStartCycleTime;

        FOR i := 0 TO AVERAGE_ARRAY_SIZE - 1 BY 1 DO
            sumAvgArray := TO_LREAL(sumAvgArray + arrLrAvgCycleTime[i]);
        END_FOR

        HMI.lrPiecePerMinute := 60000 / (sumAvgArray / AVERAGE_ARRAY_SIZE);

        HMI.PieceDoneTmp :=
            HMI.PieceDoneTmp + TO_INT(_20_AUTO.recipe.st185.xUseVerLeft) + TO_INT(_20_AUTO.recipe.st185.xUseVerRight);

        iOUT_Step := ST185_Pnp_e.DONE;
    END_IF

(***** DONE *****)
ST185_Pnp_e.DONE: (* Letzter Schritt  *)
    IF NOT xIN_AlarmAktiv THEN
        //AUTO
        IF (enIN_State = StateAUTO) AND xIN_RestartCYCL THEN
            iOUT_Step := ST185_Pnp_e.START;
            //STEP / END / LEERFAHREN restart
        ELSIF (enIN_State < StateAUTO) AND (enIN_State >= enState.StateSTEP) AND xIN_RestartCYCL THEN
            iOUT_Step := ST185_Pnp_e.START;
            //STEP / END / LEERFAHREN fertig
        ELSIF (enIN_State = StateREADY) THEN
            iOUT_Step := ST185_Pnp_e.READY;
        END_IF;
    END_IF;

(************ ERROR *************)
ST185_Pnp_e.ERROR: (* ERROR *) ;

END_CASE;

END_FUNCTION_BLOCK

// ---- POUs/20_AUTO/FileMan/FB_FileMan.TcPOU
FUNCTION_BLOCK FB_FileMan
VAR_INPUT
    sPathName   : STRING; //
    bSave       : BOOL;
    bLoad       : BOOL;
    sRefString  : POINTER TO STRING(2000);
    uiStringLen : DINT; // string length
END_VAR
VAR_OUTPUT
    bError   : BOOL;  // true when a FB is in error (all fb are mixed here)
    nErrorId : UDINT; // the error id from the fb in error (all fb are mixed here)

    bBusy : BOOL; // True when one of the local fb is busy

    currentState : INT; // current state of this FB, use it for debug
END_VAR
VAR
    fb_open  : FB_FileOpen;
    fb_write : FB_FileWrite;
    fb_read  : FB_FileRead;
    fb_close : FB_FileClose;
    hFile    : UINT; // file number holder for write operation
    state    : INT := 0;

    bOpState : INT;   //0 = saving operation, 1 = loading operation, other = error
    nMode    : DWORD; // file open monde, depending on the command

    byteRead : UDINT; //number of byte read so far
END_VAR


CASE state OF

0: (* wait for operation *)
    IF bSave THEN
        state    := 1;
        bOpState := 0;
        nMode    := FOPEN_MODEWRITE;
    ELSIF bLoad THEN
        state    := 1;
        bOpState := 1;
        nMode    := FOPEN_MODEREAD;
    END_IF

1: (* open *)
    fb_open(sNetId    := '',
            sPathName := sPathName,
            nMode     := nMode,
            ePath     := PATH_GENERIC,
            bExecute  := TRUE,
            tTimeout  := T#3S,
            bBusy     =>,
            bError    =>,
            nErrId    =>,
            hFile     => hFile);

    IF NOT fb_open.bBusy THEN
        fb_open(bExecute := FALSE);

        IF 0 = bOpState THEN
            state := 3;
        ELSIF 1 = bOpState THEN
            state    := 5;
            byteRead := 0;
        END_IF
    END_IF

3: (* write *)
    fb_write(sNetId     := '',
             hFile      := hFile,
             pWriteBuff := sRefString,
             cbWriteLen := TO_UDINT(uiStringLen),
             bExecute   := TRUE,
             tTimeout   := T#3S,
             bBusy      =>,
             bError     =>,
             nErrId     =>,
             cbWrite    =>);

    IF NOT fb_write.bBusy THEN
        fb_write(bExecute := FALSE);
        state := 10;
    END_IF

5: (* read 100 bytes *)
    IF fb_read.bEOF THEN
        state := 9;
    ELSE
        fb_read(sNetId    := '',
                hFile     := hFile,
                pReadBuff := sRefString,
                cbReadLen := TO_UDINT(uiStringLen),
                bExecute  := TRUE,
                tTimeout  :=,
                bBusy     =>,
                bError    =>,
                nErrId    =>,
                cbRead    => byteRead,
                bEOF      =>);

        state := 6;
    END_IF

6: (* open *)
    fb_read(bExecute := FALSE);
    state := 5;

9:
    state := 10;

10: (* open *)
    fb_close(sNetId   := '',
             hFile    := hFile,
             bExecute := TRUE,
             tTimeout := T#3S,
             bBusy    =>,
             bError   =>,
             nErrId   =>);

    IF NOT fb_close.bBusy AND NOT bSave AND NOT bLoad THEN
        fb_close(bExecute := FALSE);
        state := 0;
    END_IF

END_CASE

bError       := fb_open.bError OR fb_write.bError OR fb_read.bError OR fb_close.bError;
nErrorId     := fb_open.nErrId OR fb_write.nErrId OR fb_read.nErrId OR fb_close.nErrId;
bBusy        := fb_open.bBusy OR fb_write.bBusy OR fb_read.bBusy OR fb_close.bBusy;
currentState := state;

END_FUNCTION_BLOCK

// ---- POUs/20_AUTO/FileMan/FileMan.TcPOU
PROGRAM FileMan
VAR
    fb_fileMan : FB_FileMan;
    bSaveData  : BOOL := FALSE;
    bLoadData  : BOOL := TRUE;
    json_data  : STRING(20000);
	json_len : DINT;
END_VAR


fb_fileMan(sPathName    := 'D:\tmp\mover_demo.json',
           bSave        := bSaveData,
           bLoad        := bLoadData,
           sRefString   := ADR(json_data),
           bError       =>,
           nErrorId     =>,
           currentState =>);

IF fb_fileMan.currentState = 3 THEN
    IF NOT fb_fileMan.bBusy THEN
        json_len               := SaveInMemory_Recipe(json_data);
        fb_fileMan.uiStringLen := json_len;
    END_IF

ELSIF fb_fileMan.currentState = 5 THEN
    fb_fileMan.uiStringLen := 2000;

ELSIF fb_fileMan.currentState = 9 THEN
    IF NOT fb_fileMan.bBusy THEN
        ReadJsonDom(json_data);
    END_IF

ELSIF fb_fileMan.currentState = 10 THEN
    bSaveData := FALSE;
    bLoadData := FALSE;
END_IF

END_PROGRAM

// ---- POUs/20_AUTO/FileMan/SaveInMemory_Recipe.TcPOU
FUNCTION SaveInMemory_Recipe : DINT
VAR_INPUT
    sData : REFERENCE TO STRING(20000);
END_VAR
VAR
    fbJson : FB_JsonSaxWriter;

    i   : INT;
    ii  : INT;
    iii : INT;

END_VAR

fbJson.ResetDocument();
//  global object
fbJson.StartObject();

fbJson.AddKey('iStationTimeDef1');
fbJson.StartArray();

FOR i := 1 TO CONST.STATION_NUMBER BY 1 DO
    fbJson.AddDint(PERS.iStationTimeDef1[i]);
END_FOR

fbJson.EndArray();
fbJson.AddKey('iStationTimeDef2');
fbJson.StartArray();

FOR i := 1 TO CONST.STATION_NUMBER BY 1 DO
    fbJson.AddDint(PERS.iStationTimeDef2[i]);
END_FOR

fbJson.EndArray();
fbJson.addKey('recipeList');
fbJson.StartArray();

FOR i := 0 TO CONST.MAX_RECIPE_NUMBER BY 1 DO
    fbJson.StartObject();
    fbJson.addKey('linearAxis');
    fbJson.StartArray();

    FOR ii := 0 TO LinearAxis_e._max - 1 BY 1 DO
        fbJson.StartObject();
        fbJson.addKey('defProfile');
        fbJson.StartObject();
        fbJson.AddKey('lrVelocity');
        fbJson.AddLreal(PERS.recipeList[i].linearAxis[ii].defProfile.lrVelocity);
        fbJson.AddKey('lrAccel');
        fbJson.AddLreal(PERS.recipeList[i].linearAxis[ii].defProfile.lrAccel);
        fbJson.AddKey('lrDecel');
        fbJson.AddLreal(PERS.recipeList[i].linearAxis[ii].defProfile.lrDecel);
        fbJson.AddKey('lrJerk');
        fbJson.AddLreal(PERS.recipeList[i].linearAxis[ii].defProfile.lrJerk);
        fbJson.EndObject();
        fbJson.addKey('movesList');
        fbJson.StartArray();

        FOR iii := 0 TO CONST.MAX_VECTOR_LIST BY 1 DO
            fbJson.StartObject();
            fbJson.AddKey('lrVelocity');
            fbJson.AddLreal(PERS.recipeList[i].linearAxis[ii].movesList[iii].lrVelocity);
            fbJson.AddKey('lrAccel');
            fbJson.AddLreal(PERS.recipeList[i].linearAxis[ii].movesList[iii].lrAccel);
            fbJson.AddKey('lrDecel');
            fbJson.AddLreal(PERS.recipeList[i].linearAxis[ii].movesList[iii].lrDecel);
            fbJson.AddKey('lrJerk');
            fbJson.AddLreal(PERS.recipeList[i].linearAxis[ii].movesList[iii].lrJerk);
            fbJson.AddKey('lrPosition');
            fbJson.AddLreal(PERS.recipeList[i].linearAxis[ii].movesList[iii].lrPosition);
            fbJson.AddKey('TriggerType');
            fbJson.AddDint(PERS.recipeList[i].linearAxis[ii].movesList[iii].TriggerType);
            fbJson.AddKey('TriggerPos');
            fbJson.AddLreal(PERS.recipeList[i].linearAxis[ii].movesList[iii].TriggerPos);
            fbJson.AddKey('Timeout_ms');
            fbJson.AddDint(PERS.recipeList[i].linearAxis[ii].movesList[iii].Timeout_ms);
            fbJson.EndObject();
        END_FOR

        fbJson.EndArray();
        fbJson.EndObject();
    END_FOR

    fbJson.EndArray();
    fbJson.addKey('cylinder2Pos');
    fbJson.StartArray();

    FOR ii := 0 TO StationList_e._max - 1 BY 1 DO
        FOR iii := 0 TO CONST.MAX_CYLINDER_PER_STATION - 1 BY 1 DO
            fbJson.StartObject();
            fbJson.AddKey('toGS_alarm_time');
            fbJson.AddDint(PERS.recipeList[i].cylinder2Pos[ii][iii].toGS_alarm_time);
            fbJson.AddKey('toAS_alarm_time');
            fbJson.AddDint(PERS.recipeList[i].cylinder2Pos[ii][iii].toAS_alarm_time);
            fbJson.AddKey('toGS_wait_time');
            fbJson.AddDint(PERS.recipeList[i].cylinder2Pos[ii][iii].toGS_wait_time);
            fbJson.AddKey('toAS_wait_time');
            fbJson.AddDint(PERS.recipeList[i].cylinder2Pos[ii][iii].toAS_wait_time);
            fbJson.EndObject();
        END_FOR
    END_FOR

    fbJson.EndArray();
    fbJson.AddKey('stationOffsets');
    fbJson.StartArray();

    FOR ii := 0 TO CONST.STATION_NUMBER - 1 BY 1 DO
        fbJson.AddLreal(PERS.recipeList[i].stationOffsets[ii]);
    END_FOR

    fbJson.EndArray();
    fbJson.addKey('st110');
    fbJson.StartObject();
    fbJson.AddKey('xUseVerLeft');
    fbJson.AddBool(PERS.recipeList[i].st110.xUseVerLeft);
    fbJson.AddKey('xUseVerRight');
    fbJson.AddBool(PERS.recipeList[i].st110.xUseVerRight);
    fbJson.addKey('FeederConfig');
    fbJson.StartObject();
    fbJson.AddKey('InFilterDelay');
    fbJson.AddDint(PERS.recipeList[i].st110.FeederConfig.InFilterDelay);
    fbJson.AddKey('StartDelay');
    fbJson.AddDint(PERS.recipeList[i].st110.FeederConfig.StartDelay);
    fbJson.AddKey('StopDelay');
    fbJson.AddDint(PERS.recipeList[i].st110.FeederConfig.StopDelay);
    fbJson.AddKey('EmptyDelay');
    fbJson.AddDint(PERS.recipeList[i].st110.FeederConfig.EmptyDelay);
    fbJson.EndObject();
    fbJson.EndObject();
    fbJson.addKey('st115');
    fbJson.StartObject();
    fbJson.AddKey('xUseVerLeft');
    fbJson.AddBool(PERS.recipeList[i].st115.xUseVerLeft);
    fbJson.AddKey('xUseVerRight');
    fbJson.AddBool(PERS.recipeList[i].st115.xUseVerRight);
    fbJson.addKey('FeederConfig');
    fbJson.StartObject();
    fbJson.AddKey('InFilterDelay');
    fbJson.AddDint(PERS.recipeList[i].st115.FeederConfig.InFilterDelay);
    fbJson.AddKey('StartDelay');
    fbJson.AddDint(PERS.recipeList[i].st115.FeederConfig.StartDelay);
    fbJson.AddKey('StopDelay');
    fbJson.AddDint(PERS.recipeList[i].st115.FeederConfig.StopDelay);
    fbJson.AddKey('EmptyDelay');
    fbJson.AddDint(PERS.recipeList[i].st115.FeederConfig.EmptyDelay);
    fbJson.EndObject();
    fbJson.EndObject();
    fbJson.addKey('st120');
    fbJson.StartObject();
    fbJson.AddKey('xUseVerLeft');
    fbJson.AddBool(PERS.recipeList[i].st120.xUseVerLeft);
    fbJson.AddKey('xUseVerRight');
    fbJson.AddBool(PERS.recipeList[i].st120.xUseVerRight);
    fbJson.addKey('FeederConfigLeft');
    fbJson.StartObject();
    fbJson.AddKey('InFilterDelay');
    fbJson.AddDint(PERS.recipeList[i].st120.FeederConfigLeft.InFilterDelay);
    fbJson.AddKey('StartDelay');
    fbJson.AddDint(PERS.recipeList[i].st120.FeederConfigLeft.StartDelay);
    fbJson.AddKey('StopDelay');
    fbJson.AddDint(PERS.recipeList[i].st120.FeederConfigLeft.StopDelay);
    fbJson.AddKey('EmptyDelay');
    fbJson.AddDint(PERS.recipeList[i].st120.FeederConfigLeft.EmptyDelay);
    fbJson.EndObject();
    fbJson.addKey('FeederConfigRight');
    fbJson.StartObject();
    fbJson.AddKey('InFilterDelay');
    fbJson.AddDint(PERS.recipeList[i].st120.FeederConfigRight.InFilterDelay);
    fbJson.AddKey('StartDelay');
    fbJson.AddDint(PERS.recipeList[i].st120.FeederConfigRight.StartDelay);
    fbJson.AddKey('StopDelay');
    fbJson.AddDint(PERS.recipeList[i].st120.FeederConfigRight.StopDelay);
    fbJson.AddKey('EmptyDelay');
    fbJson.AddDint(PERS.recipeList[i].st120.FeederConfigRight.EmptyDelay);
    fbJson.EndObject();
    fbJson.EndObject();
    fbJson.addKey('st125');
    fbJson.StartObject();
    fbJson.addKey('ST125_Recipe_t');
    fbJson.StartObject();
    fbJson.AddKey('xUseVerLeft');
    fbJson.AddBool(PERS.recipeList[i].st125.xUseVerLeft);
    fbJson.AddKey('xUseVerRight');
    fbJson.AddBool(PERS.recipeList[i].st125.xUseVerRight);
    fbJson.addKey('FeederConfig');
    fbJson.StartObject();
    fbJson.AddKey('InFilterDelay');
    fbJson.AddDint(PERS.recipeList[i].st125.FeederConfig.InFilterDelay);
    fbJson.AddKey('StartDelay');
    fbJson.AddDint(PERS.recipeList[i].st125.FeederConfig.StartDelay);
    fbJson.AddKey('StopDelay');
    fbJson.AddDint(PERS.recipeList[i].st125.FeederConfig.StopDelay);
    fbJson.AddKey('EmptyDelay');
    fbJson.AddDint(PERS.recipeList[i].st125.FeederConfig.EmptyDelay);
    fbJson.EndObject();
    fbJson.EndObject();
    fbJson.EndObject();
    fbJson.addKey('st145');
    fbJson.StartObject();
    fbJson.addKey('ST145_Recipe_t');
    fbJson.StartObject();
    fbJson.AddKey('xUseVerLeft');
    fbJson.AddBool(PERS.recipeList[i].st145.xUseVerLeft);
    fbJson.AddKey('xUseVerRight');
    fbJson.AddBool(PERS.recipeList[i].st145.xUseVerRight);
    fbJson.addKey('FeederConfig');
    fbJson.StartObject();
    fbJson.AddKey('InFilterDelay');
    fbJson.AddDint(PERS.recipeList[i].st145.FeederConfig.InFilterDelay);
    fbJson.AddKey('StartDelay');
    fbJson.AddDint(PERS.recipeList[i].st145.FeederConfig.StartDelay);
    fbJson.AddKey('StopDelay');
    fbJson.AddDint(PERS.recipeList[i].st145.FeederConfig.StopDelay);
    fbJson.AddKey('EmptyDelay');
    fbJson.AddDint(PERS.recipeList[i].st145.FeederConfig.EmptyDelay);
    fbJson.EndObject();
    fbJson.EndObject();
    fbJson.EndObject();
    fbJson.addKey('st180');
    fbJson.StartObject();
    fbJson.AddKey('xUseVerLeft');
    fbJson.AddBool(PERS.recipeList[i].st180.xUseVerLeft);
    fbJson.AddKey('xUseVerRight');
    fbJson.AddBool(PERS.recipeList[i].st180.xUseVerRight);
    fbJson.EndObject();
    fbJson.EndObject();
END_FOR

fbJson.EndArray();
fbJson.AddKey('iRecipeCurrent');
fbJson.AddDint(PERS.iRecipeCurrent);

// end global object
fbJson.EndObject();
// end of file
SaveInMemory_Recipe := TO_DINT(fbJson.CopyDocument(sData, fbJson.GetDocumentLength()));
fbJson.ResetDocument();

END_FUNCTION

// ---- POUs/20_AUTO/FileMan/ReadJsonDom.TcPOU
FUNCTION ReadJsonDom : BOOL
VAR_INPUT
END_VAR
VAR
    fb_json : FB_JsonDomParser;

    json_head              : SJsonValue;
    json_value             : SJsonValue;
    json_iStationTimeDef1  : SJsonValue;
    json_iStationTimeDef2  : SJsonValue;
    json_recipeList        : SJsonValue;
    json_linearAxis        : SJsonValue;
    json_defProfile        : SJsonValue;
    json_movesList         : SJsonValue;
    json_cylinder2Pos      : SJsonValue;
    json_stationOffsets    : SJsonValue;
    json_st110             : SJsonValue;
    json_FeederConfig      : SJsonValue;
    json_st115             : SJsonValue;
    json_st120             : SJsonValue;
    json_FeederConfigLeft  : SJsonValue;
    json_FeederConfigRight : SJsonValue;
    json_st125             : SJsonValue;
    json_st145             : SJsonValue;
    json_st180             : SJsonValue;
    json_i                 : SJsonValue;
    json_ii                : SJsonValue;
    json_iii               : SJsonValue;

    i   : INT;
    ii  : INT;
    iii : INT;

END_VAR
VAR_IN_OUT
    sMessage : STRING(10000);
END_VAR

json_head := fb_json.ParseDocument(sMessage);

IF fb_json.HasMember(json_head, 'iStationTimeDef1') THEN
    json_iStationTimeDef1 := fb_json.FindMember(json_head, 'iStationTimeDef1');

    IF fb_json.IsArray(json_iStationTimeDef1) THEN
        FOR i := 0 TO MIN(TO_INT(fb_json.GetArraySize(json_iStationTimeDef1)) - 1, CONST.STATION_NUMBER - 1) BY 1 DO
            json_i                       := fb_json.GetArrayValueByIdx(json_iStationTimeDef1, TO_UDINT(i));
            PERS.iStationTimeDef1[i + 1] := TO_DINT(fb_json.GetInt(json_i));
        END_FOR
    END_IF
END_IF

IF fb_json.HasMember(json_head, 'iStationTimeDef2') THEN
    json_iStationTimeDef2 := fb_json.FindMember(json_head, 'iStationTimeDef2');

    IF fb_json.IsArray(json_iStationTimeDef2) THEN
        FOR i := 0 TO MIN(TO_INT(fb_json.GetArraySize(json_iStationTimeDef2)) - 1, CONST.STATION_NUMBER - 1) BY 1 DO
            json_i                       := fb_json.GetArrayValueByIdx(json_iStationTimeDef2, TO_UDINT(i));
            PERS.iStationTimeDef2[i + 1] := TO_DINT(fb_json.GetInt(json_i));
        END_FOR
    END_IF
END_IF

IF fb_json.HasMember(json_head, 'recipeList') THEN
    json_recipeList := fb_json.FindMember(json_head, 'recipeList');

    IF fb_json.IsArray(json_recipeList) THEN
        FOR i := 0 TO MIN(TO_INT(fb_json.GetArraySize(json_recipeList)) - 1, CONST.MAX_RECIPE_NUMBER - 0) BY 1 DO
            json_i := fb_json.GetArrayValueByIdx(json_recipeList, TO_UDINT(i));

            IF fb_json.HasMember(json_i, 'linearAxis') THEN
                json_linearAxis := fb_json.FindMember(json_i, 'linearAxis');

                IF fb_json.IsArray(json_linearAxis) THEN
                    FOR ii := 0 TO MIN(TO_INT(fb_json.GetArraySize(json_linearAxis)) - 1, LinearAxis_e._max - 1 - 0) BY
                        1 DO
                        json_ii := fb_json.GetArrayValueByIdx(json_linearAxis, TO_UDINT(ii));

                        IF fb_json.HasMember(json_ii, 'defProfile') THEN
                            json_defProfile := fb_json.FindMember(json_ii, 'defProfile');

                            IF fb_json.HasMember(json_defProfile, 'lrVelocity') THEN
                                json_value := fb_json.FindMember(json_defProfile, 'lrVelocity');
                                PERS.recipeList[i + 0].linearAxis[ii + 0].defProfile.lrVelocity
                                    := TO_REAL(fb_json.GetDouble(json_value));
                            END_IF

                            IF fb_json.HasMember(json_defProfile, 'lrAccel') THEN
                                json_value := fb_json.FindMember(json_defProfile, 'lrAccel');
                                PERS.recipeList[i + 0].linearAxis[ii + 0].defProfile.lrAccel
                                    := TO_REAL(fb_json.GetDouble(json_value));
                            END_IF

                            IF fb_json.HasMember(json_defProfile, 'lrDecel') THEN
                                json_value := fb_json.FindMember(json_defProfile, 'lrDecel');
                                PERS.recipeList[i + 0].linearAxis[ii + 0].defProfile.lrDecel
                                    := TO_REAL(fb_json.GetDouble(json_value));
                            END_IF

                            IF fb_json.HasMember(json_defProfile, 'lrJerk') THEN
                                json_value := fb_json.FindMember(json_defProfile, 'lrJerk');
                                PERS.recipeList[i + 0].linearAxis[ii + 0].defProfile.lrJerk
                                    := TO_REAL(fb_json.GetDouble(json_value));
                            END_IF
                        END_IF

                        IF fb_json.HasMember(json_ii, 'movesList') THEN
                            json_movesList := fb_json.FindMember(json_ii, 'movesList');

                            IF fb_json.IsArray(json_movesList) THEN
                                FOR iii := 0 TO
                                    MIN(TO_INT(fb_json.GetArraySize(json_movesList)) - 1, CONST.MAX_VECTOR_LIST - 0) BY
                                    1 DO
                                    json_iii := fb_json.GetArrayValueByIdx(json_movesList, TO_UDINT(iii));

                                    IF fb_json.HasMember(json_iii, 'lrVelocity') THEN
                                        json_value := fb_json.FindMember(json_iii, 'lrVelocity');
                                        PERS.recipeList[i + 0].linearAxis[ii + 0].movesList[iii + 0].lrVelocity
                                            := TO_REAL(fb_json.GetDouble(json_value));
                                    END_IF

                                    IF fb_json.HasMember(json_iii, 'lrAccel') THEN
                                        json_value := fb_json.FindMember(json_iii, 'lrAccel');
                                        PERS.recipeList[i + 0].linearAxis[ii + 0].movesList[iii + 0].lrAccel
                                            := TO_REAL(fb_json.GetDouble(json_value));
                                    END_IF

                                    IF fb_json.HasMember(json_iii, 'lrDecel') THEN
                                        json_value := fb_json.FindMember(json_iii, 'lrDecel');
                                        PERS.recipeList[i + 0].linearAxis[ii + 0].movesList[iii + 0].lrDecel
                                            := TO_REAL(fb_json.GetDouble(json_value));
                                    END_IF

                                    IF fb_json.HasMember(json_iii, 'lrJerk') THEN
                                        json_value := fb_json.FindMember(json_iii, 'lrJerk');
                                        PERS.recipeList[i + 0].linearAxis[ii + 0].movesList[iii + 0].lrJerk
                                            := TO_REAL(fb_json.GetDouble(json_value));
                                    END_IF

                                    IF fb_json.HasMember(json_iii, 'lrPosition') THEN
                                        json_value := fb_json.FindMember(json_iii, 'lrPosition');
                                        PERS.recipeList[i + 0].linearAxis[ii + 0].movesList[iii + 0].lrPosition
                                            := TO_LREAL(fb_json.GetDouble(json_value));
                                    END_IF

                                    IF fb_json.HasMember(json_iii, 'TriggerType') THEN
                                        json_value := fb_json.FindMember(json_iii, 'TriggerType');
                                        PERS.recipeList[i + 0].linearAxis[ii + 0].movesList[iii + 0].TriggerType
                                            := TO_INT(fb_json.GetInt(json_value));
                                    END_IF

                                    IF fb_json.HasMember(json_iii, 'TriggerPos') THEN
                                        json_value := fb_json.FindMember(json_iii, 'TriggerPos');
                                        PERS.recipeList[i + 0].linearAxis[ii + 0].movesList[iii + 0].TriggerPos
                                            := TO_LREAL(fb_json.GetDouble(json_value));
                                    END_IF

                                    IF fb_json.HasMember(json_iii, 'Timeout_ms') THEN
                                        json_value := fb_json.FindMember(json_iii, 'Timeout_ms');
                                        PERS.recipeList[i + 0].linearAxis[ii + 0].movesList[iii + 0].Timeout_ms
                                            := TO_DINT(fb_json.GetInt(json_value));
                                    END_IF
                                END_FOR
                            END_IF
                        END_IF
                    END_FOR
                END_IF
            END_IF

            IF fb_json.HasMember(json_i, 'cylinder2Pos') THEN
                json_cylinder2Pos := fb_json.FindMember(json_i, 'cylinder2Pos');

                IF fb_json.IsArray(json_cylinder2Pos) THEN
                    FOR ii := 0 TO MIN(TO_INT(fb_json.GetArraySize(json_cylinder2Pos)) - 1, StationList_e._max - 1) BY
                        1 DO
                        json_ii := fb_json.GetArrayValueByIdx(json_cylinder2Pos, TO_UDINT(ii));

                        IF fb_json.IsArray(json_ii) THEN
                            FOR iii := 0 TO
                                MIN(TO_INT(fb_json.GetArraySize(json_ii)) - 1, CONST.MAX_CYLINDER_PER_STATION - 1) BY
                                1 DO
                                json_iii := fb_json.GetArrayValueByIdx(json_ii, TO_UDINT(iii));

                                IF fb_json.HasMember(json_iii, 'toGS_alarm_time') THEN
                                    json_value := fb_json.FindMember(json_iii, 'toGS_alarm_time');
                                    PERS.recipeList[i + 0].cylinder2Pos[ii + 0][iii + 0].toGS_alarm_time
                                        := TO_DINT(fb_json.GetInt(json_value));
                                END_IF

                                IF fb_json.HasMember(json_iii, 'toAS_alarm_time') THEN
                                    json_value := fb_json.FindMember(json_iii, 'toAS_alarm_time');
                                    PERS.recipeList[i + 0].cylinder2Pos[ii + 0][iii + 0].toAS_alarm_time
                                        := TO_DINT(fb_json.GetInt(json_value));
                                END_IF

                                IF fb_json.HasMember(json_iii, 'toGS_wait_time') THEN
                                    json_value := fb_json.FindMember(json_iii, 'toGS_wait_time');
                                    PERS.recipeList[i + 0].cylinder2Pos[ii + 0][iii + 0].toGS_wait_time
                                        := TO_DINT(fb_json.GetInt(json_value));
                                END_IF

                                IF fb_json.HasMember(json_iii, 'toAS_wait_time') THEN
                                    json_value := fb_json.FindMember(json_iii, 'toAS_wait_time');
                                    PERS.recipeList[i + 0].cylinder2Pos[ii + 0][iii + 0].toAS_wait_time
                                        := TO_DINT(fb_json.GetInt(json_value));
                                END_IF
                            END_FOR
                        END_IF
                    END_FOR
                END_IF

                IF fb_json.HasMember(json_i, 'stationOffsets') THEN
                    json_stationOffsets := fb_json.FindMember(json_i, 'stationOffsets');

                    IF fb_json.IsArray(json_stationOffsets) THEN
                        FOR ii := 0 TO
                            MIN(TO_INT(fb_json.GetArraySize(json_stationOffsets)) - 1, CONST.STATION_NUMBER - 1 - 0) BY
                            1 DO
                            json_ii := fb_json.GetArrayValueByIdx(json_stationOffsets, TO_UDINT(ii));
                            PERS.recipeList[i + 0].stationOffsets[ii + 0]
                                := TO_REAL(fb_json.GetDouble(json_ii));
                        END_FOR
                    END_IF
                END_IF

                IF fb_json.HasMember(json_i, 'st110') THEN
                    json_st110 := fb_json.FindMember(json_i, 'st110');

                    IF fb_json.HasMember(json_st110, 'xUseVerLeft') THEN
                        json_value                               := fb_json.FindMember(json_st110, 'xUseVerLeft');
                        PERS.recipeList[i + 0].st110.xUseVerLeft := TO_BOOL(fb_json.GetBool(json_value));
                    END_IF

                    IF fb_json.HasMember(json_st110, 'xUseVerRight') THEN
                        json_value                                := fb_json.FindMember(json_st110, 'xUseVerRight');
                        PERS.recipeList[i + 0].st110.xUseVerRight := TO_BOOL(fb_json.GetBool(json_value));
                    END_IF

                    IF fb_json.HasMember(json_st110, 'FeederConfig') THEN
                        json_FeederConfig := fb_json.FindMember(json_st110, 'FeederConfig');

